LIN {X 0,Y 229.59,Z 265.503,A -85,B 0,C 180,E1 -20151.196,E2 -20151.196} C_VEL
LIN {X 0,Y 229.22,Z 263.63,A -85,B 0,C 180,E1 -20152.955,E2 -20152.955} C_VEL
LIN {X 0,Y 228.29,Z 260.05,A -85,B 0,C 180,E1 -20156.691,E2 -20156.691} C_VEL
LIN {X 0,Y 228.555,Z 260.016,A -85,B 0,C 180,E1 -20158.238,E2 -20158.238} C_VEL
LIN {X 0,Y 228.555,Z 260.014,A -85,B 0,C 180,E1 -20161.762,E2 -20161.762} C_VEL
LIN {X 0,Y 228.313,Z 260.047,A -85,B 0,C 180,E1 -20167.073,E2 -20167.073} C_VEL
LIN {X 0,Y 228.147,Z 260.063,A -85,B 0,C 180,E1 -20170.651,E2 -20170.651} C_VEL
LIN {X 0,Y 228.066,Z 260.074,A -85,B 0,C 180,E1 -20174.272,E2 -20174.272} C_VEL
LIN {X 0,Y 228.004,Z 260.082,A -85,B 0,C 180,E1 -20177.953,E2 -20177.953} C_VEL
LIN {X 0,Y 227.918,Z 260.094,A -85,B 0,C 180,E1 -20182.321,E2 -20182.321} C_VEL
LIN {X 0,Y 227.944,Z 260.087,A -85,B 0,C 180,E1 -20186.603,E2 -20186.603} C_VEL
LIN {X 0,Y 227.91,Z 260.093,A -85,B 0,C 180,E1 -20190.296,E2 -20190.296} C_VEL
LIN {X 0,Y 227.889,Z 260.097,A -85,B 0,C 180,E1 -20193.718,E2 -20193.718} C_VEL
LIN {X 0,Y 227.86,Z 260.1,A -85,B 0,C 180,E1 -20198.088,E2 -20198.088} C_VEL
LIN {X 0,Y 227.945,Z 260.09,A -85,B 0,C 180,E1 -20202.711,E2 -20202.711} C_VEL
LIN {X 0,Y 228.096,Z 260.26,A -85,B 0,C 180,E1 -20204.606,E2 -20204.606} C_VEL
LIN {X 0,Y 228.501,Z 262.622,A -85,B 0,C 180,E1 -20206.87,E2 -20206.87} C_VEL
LIN {X 0,Y 230.282,Z 270.126,A -85,B 0,C 180,E1 -20211.134,E2 -20211.134} C_VEL
LIN {X 0,Y 230.396,Z 272.05,A -85,B 0,C 180,E1 -20211.985,E2 -20211.985} C_VEL
LIN {X 0,Y 229.973,Z 274.309,A -85,B 0,C 180,E1 -20212.782,E2 -20212.782} C_VEL
LIN {X 0,Y 228.181,Z 279.291,A -85,B 0,C 180,E1 -20214.258,E2 -20214.258} C_VEL
LIN {X 0,Y 225.385,Z 287.27,A -85,B 0,C 180,E1 -20216.474,E2 -20216.474} C_VEL
LIN {X 0,Y 225.099,Z 289.77,A -85,B 0,C 180,E1 -20217.278,E2 -20217.278} C_VEL
LIN {X 0,Y 225.285,Z 297.17,A -85,B 0,C 180,E1 -20219.681,E2 -20219.681} C_VEL
LIN {X 0,Y 228.899,Z 309.726,A -85,B 0,C 180,E1 -20221.127,E2 -20221.127} C_VEL
LIN {X 0,Y 230.455,Z 318.269,A -85,B 0,C 180,E1 -20222.176,E2 -20222.176} C_VEL
LIN {X 0,Y 230.206,Z 328.596,A -85,B 0,C 180,E1 -20223.391,E2 -20223.391} C_VEL
LIN {X 0,Y 229.898,Z 337.162,A -85,B 0,C 180,E1 -20224.661,E2 -20224.661} C_VEL
LIN {X 0,Y 229.393,Z 343.849,A -85,B 0,C 180,E1 -20225.809,E2 -20225.809} C_VEL
LIN {X 0,Y 227.633,Z 351.72,A -85,B 0,C 180,E1 -20227.299,E2 -20227.299} C_VEL
LIN {X 0,Y 225.585,Z 359.464,A -85,B 0,C 180,E1 -20229.101,E2 -20229.101} C_VEL
LIN {X 0,Y 224.128,Z 365.266,A -85,B 0,C 180,E1 -20230.777,E2 -20230.777} C_VEL
LIN {X 0,Y 222.433,Z 371.587,A -85,B 0,C 180,E1 -20233.007,E2 -20233.007} C_VEL
LIN {X 0,Y 220.953,Z 376.675,A -85,B 0,C 180,E1 -20235.259,E2 -20235.259} C_VEL
LIN {X 0,Y 219.787,Z 381.363,A -85,B 0,C 180,E1 -20238.004,E2 -20238.004} C_VEL
LIN {X 0,Y 219.081,Z 384.647,A -85,B 0,C 180,E1 -20240.77,E2 -20240.77} C_VEL
LIN {X 0,Y 218.848,Z 386.24,A -85,B 0,C 180,E1 -20242.62,E2 -20242.62} C_VEL
LIN {X 0,Y 218.718,Z 387.462,A -85,B 0,C 180,E1 -20244.946,E2 -20244.946} C_VEL
LIN {X 0,Y 218.899,Z 387.78,A -85,B 0,C 180,E1 -20248.16,E2 -20248.16} C_VEL
LIN {X 0,Y 219.007,Z 387.299,A -85,B 0,C 180,E1 -20250,E2 -20250} C_VEL
LIN {X 0,Y 219.025,Z 386.314,A -85,B 0,C 180,E1 -20251.839,E2 -20251.839} C_VEL
LIN {X 0,Y 218.977,Z 384.863,A -85,B 0,C 180,E1 -20253.681,E2 -20253.681} C_VEL
LIN {X 0,Y 218.888,Z 386.594,A -85,B 0,C 180,E1 -20257.379,E2 -20257.379} C_VEL
LIN {X 0,Y 219.575,Z 386.929,A -85,B 0,C 180,E1 -20261.072,E2 -20261.072} C_VEL
LIN {X 0,Y 221.154,Z 385.921,A -85,B 0,C 180,E1 -20264.728,E2 -20264.728} C_VEL
LIN {X 0,Y 224.036,Z 383.598,A -85,B 0,C 180,E1 -20268.283,E2 -20268.283} C_VEL
LIN {X 0,Y 227.711,Z 379.914,A -85,B 0,C 180,E1 -20271.738,E2 -20271.738} C_VEL
LIN {X 0,Y 232.452,Z 374.872,A -85,B 0,C 180,E1 -20275.042,E2 -20275.042} C_VEL
LIN {X 0,Y 238.466,Z 368.336,A -85,B 0,C 180,E1 -20278.135,E2 -20278.135} C_VEL
LIN {X 0,Y 245.331,Z 360.115,A -85,B 0,C 180,E1 -20281.041,E2 -20281.041} C_VEL
LIN {X 0,Y 247.83,Z 356.7,A -85,B 0,C 180,E1 -20282.122,E2 -20282.122} C_VEL
LIN {X 0,Y 250.643,Z 351.199,A -85,B 0,C 180,E1 -20284.112,E2 -20284.112} C_VEL
LIN {X 0,Y 253.194,Z 344.707,A -85,B 0,C 180,E1 -20286.639,E2 -20286.639} C_VEL
LIN {X 0,Y 255.221,Z 338.662,A -85,B 0,C 180,E1 -20289.298,E2 -20289.298} C_VEL
LIN {X 0,Y 256.199,Z 335.187,A -85,B 0,C 180,E1 -20291.176,E2 -20291.176} C_VEL
LIN {X 0,Y 256.438,Z 333.729,A -85,B 0,C 180,E1 -20292.271,E2 -20292.271} C_VEL
LIN {X 0,Y 256.512,Z 331.788,A -85,B 0,C 180,E1 -20294.573,E2 -20294.573} C_VEL
LIN {X 0,Y 256.711,Z 330.528,A -85,B 0,C 180,E1 -20297.663,E2 -20297.663} C_VEL
LIN {X 0,Y 257.03,Z 330.502,A -85,B 0,C 180,E1 -20299.962,E2 -20299.962} C_VEL
LIN {X 0,Y 257.237,Z 331.647,A -85,B 0,C 180,E1 -20302.403,E2 -20302.403} C_VEL
LIN {X 0,Y 257.278,Z 333.985,A -85,B 0,C 180,E1 -20305.036,E2 -20305.036} C_VEL
LIN {X 0,Y 256.953,Z 336.363,A -85,B 0,C 180,E1 -20306.837,E2 -20306.837} C_VEL
LIN {X 0,Y 256.352,Z 339.157,A -85,B 0,C 180,E1 -20308.608,E2 -20308.608} C_VEL
LIN {X 0,Y 255.812,Z 340.134,A -85,B 0,C 180,E1 -20309.005,E2 -20309.005} C_VEL
LIN {X 0,Y 249.23,Z 347.794,A -85,B 0,C 180,E1 -20311.355,E2 -20311.355} C_VEL
LIN {X 0,Y 244.122,Z 353.199,A -85,B 0,C 180,E1 -20313.498,E2 -20313.498} C_VEL
LIN {X 0,Y 237.984,Z 358.947,A -85,B 0,C 180,E1 -20316.505,E2 -20316.505} C_VEL
LIN {X 0,Y 233.908,Z 362.242,A -85,B 0,C 180,E1 -20318.866,E2 -20318.866} C_VEL
LIN {X 0,Y 229.169,Z 365.414,A -85,B 0,C 180,E1 -20322.141,E2 -20322.141} C_VEL
LIN {X 0,Y 225.4,Z 367.13,A -85,B 0,C 180,E1 -20325.556,E2 -20325.556} C_VEL
LIN {X 0,Y 223.711,Z 367.493,A -85,B 0,C 180,E1 -20327.296,E2 -20327.296} C_VEL
LIN {X 0,Y 221.617,Z 367.146,A -85,B 0,C 180,E1 -20330.877,E2 -20330.877} C_VEL
LIN {X 0,Y 220.129,Z 365.421,A -85,B 0,C 180,E1 -20334.504,E2 -20334.504} C_VEL
LIN {X 0,Y 219.102,Z 362.21,A -85,B 0,C 180,E1 -20338.162,E2 -20338.162} C_VEL
LIN {X 0,Y 218.911,Z 357.473,A -85,B 0,C 180,E1 -20341.84,E2 -20341.84} C_VEL
LIN {X 0,Y 218.884,Z 352.437,A -85,B 0,C 180,E1 -20344.746,E2 -20344.746} C_VEL
LIN {X 0,Y 219.258,Z 345.516,A -85,B 0,C 180,E1 -20347.903,E2 -20347.903} C_VEL
LIN {X 0,Y 219.791,Z 338.239,A -85,B 0,C 180,E1 -20350.595,E2 -20350.595} C_VEL
LIN {X 0,Y 220.562,Z 329.134,A -85,B 0,C 180,E1 -20353.357,E2 -20353.357} C_VEL
LIN {X 0,Y 221.665,Z 318.962,A -85,B 0,C 180,E1 -20355.871,E2 -20355.871} C_VEL
LIN {X 0,Y 222.811,Z 307.745,A -85,B 0,C 180,E1 -20358.149,E2 -20358.149} C_VEL
LIN {X 0,Y 224.156,Z 295.298,A -85,B 0,C 180,E1 -20360.175,E2 -20360.175} C_VEL
LIN {X 0,Y 224.4,Z 292.082,A -85,B 0,C 180,E1 -20360.631,E2 -20360.631} C_VEL
LIN {X 0,Y 222.196,Z 278.963,A -85,B 0,C 180,E1 -20362.307,E2 -20362.307} C_VEL
LIN {X 0,Y 219.935,Z 265.484,A -85,B 0,C 180,E1 -20363.663,E2 -20363.663} C_VEL
LIN {X 0,Y 219.354,Z 261.163,A -85,B 0,C 180,E1 -20364.07,E2 -20364.07} C_VEL
LIN {X 0,Y 219.832,Z 261.101,A -85,B 0,C 180,E1 -20368.656,E2 -20368.656} C_VEL
LIN {X 0,Y 220.291,Z 261.043,A -85,B 0,C 180,E1 -20372.845,E2 -20372.845} C_VEL
LIN {X 0,Y 220.71,Z 260.994,A -85,B 0,C 180,E1 -20377.243,E2 -20377.243} C_VEL
LIN {X 0,Y 220.775,Z 260.981,A -85,B 0,C 180,E1 -20380.181,E2 -20380.181} C_VEL
LIN {X 0,Y 220.769,Z 260.985,A -85,B 0,C 180,E1 -20384.456,E2 -20384.456} C_VEL
LIN {X 0,Y 220.761,Z 260.983,A -85,B 0,C 180,E1 -20388.045,E2 -20388.045} C_VEL
LIN {X 0,Y 220.827,Z 260.978,A -85,B 0,C 180,E1 -20392.793,E2 -20392.793} C_VEL
LIN {X 0,Y 220.815,Z 260.978,A -85,B 0,C 180,E1 -20397.243,E2 -20397.243} C_VEL
LIN {X 0,Y 220.809,Z 260.979,A -85,B 0,C 180,E1 -20401.482,E2 -20401.482} C_VEL
LIN {X 0,Y 220.854,Z 260.973,A -85,B 0,C 180,E1 -20405.563,E2 -20405.563} C_VEL
LIN {X 0,Y 220.891,Z 260.969,A -85,B 0,C 180,E1 -20409.513,E2 -20409.513} C_VEL
LIN {X 0,Y 221.02,Z 260.948,A -85,B 0,C 180,E1 -20413.37,E2 -20413.37} C_VEL
LIN {X 0,Y 221.085,Z 260.946,A -85,B 0,C 180,E1 -20419.004,E2 -20419.004} C_VEL
LIN {X 0,Y 221.245,Z 260.927,A -85,B 0,C 180,E1 -20422.7,E2 -20422.7} C_VEL
LIN {X 0,Y 221.488,Z 260.898,A -85,B 0,C 180,E1 -20429.091,E2 -20429.091} C_VEL
LIN {X 0,Y 221.548,Z 261.06,A -85,B 0,C 180,E1 -20430,E2 -20430} C_VEL
LIN {X 0,Y 221.881,Z 264.958,A -85,B 0,C 180,E1 -20432.723,E2 -20432.723} C_VEL
LIN {X 0,Y 221.791,Z 268.968,A -85,B 0,C 180,E1 -20435.455,E2 -20435.455} C_VEL
LIN {X 0,Y 221.3,Z 275.909,A -85,B 0,C 180,E1 -20440.102,E2 -20440.102} C_VEL
LIN {X 0,Y 220.873,Z 282.219,A -85,B 0,C 180,E1 -20444.276,E2 -20444.276} C_VEL
LIN {X 0,Y 222.943,Z 293.041,A -85,B 0,C 180,E1 -20445.191,E2 -20445.191} C_VEL
LIN {X 0,Y 224.555,Z 303.788,A -85,B 0,C 180,E1 -20446.36,E2 -20446.36} C_VEL
LIN {X 0,Y 225.741,Z 313.184,A -85,B 0,C 180,E1 -20447.671,E2 -20447.671} C_VEL
LIN {X 0,Y 224.619,Z 322.5,A -85,B 0,C 180,E1 -20449.179,E2 -20449.179} C_VEL
LIN {X 0,Y 223.529,Z 330.156,A -85,B 0,C 180,E1 -20450.714,E2 -20450.714} C_VEL
LIN {X 0,Y 222.436,Z 337.562,A -85,B 0,C 180,E1 -20452.537,E2 -20452.537} C_VEL
LIN {X 0,Y 221.49,Z 343.632,A -85,B 0,C 180,E1 -20454.362,E2 -20454.362} C_VEL
LIN {X 0,Y 220.462,Z 350.189,A -85,B 0,C 180,E1 -20456.797,E2 -20456.797} C_VEL
LIN {X 0,Y 219.652,Z 355.46,A -85,B 0,C 180,E1 -20459.4,E2 -20459.4} C_VEL
LIN {X 0,Y 219.037,Z 359.351,A -85,B 0,C 180,E1 -20461.966,E2 -20461.966} C_VEL
LIN {X 0,Y 218.799,Z 361.066,A -85,B 0,C 180,E1 -20463.369,E2 -20463.369} C_VEL
LIN {X 0,Y 218.61,Z 362.855,A -85,B 0,C 180,E1 -20465.357,E2 -20465.357} C_VEL
LIN {X 0,Y 218.638,Z 364.15,A -85,B 0,C 180,E1 -20467.643,E2 -20467.643} C_VEL
LIN {X 0,Y 218.886,Z 364.671,A -85,B 0,C 180,E1 -20469.953,E2 -20469.953} C_VEL
LIN {X 0,Y 219.44,Z 364.308,A -85,B 0,C 180,E1 -20472.555,E2 -20472.555} C_VEL
LIN {X 0,Y 220.372,Z 362.667,A -85,B 0,C 180,E1 -20475.443,E2 -20475.443} C_VEL
LIN {X 0,Y 221.05,Z 361.34,A -85,B 0,C 180,E1 -20476.992,E2 -20476.992} C_VEL
LIN {X 0,Y 222.318,Z 358.407,A -85,B 0,C 180,E1 -20479.349,E2 -20479.349} C_VEL
LIN {X 0,Y 223.916,Z 354.408,A -85,B 0,C 180,E1 -20481.69,E2 -20481.69} C_VEL
LIN {X 0,Y 225.719,Z 349.165,A -85,B 0,C 180,E1 -20484.051,E2 -20484.051} C_VEL
LIN {X 0,Y 227.969,Z 342.698,A -85,B 0,C 180,E1 -20486.295,E2 -20486.295} C_VEL
LIN {X 0,Y 230.573,Z 334.068,A -85,B 0,C 180,E1 -20488.59,E2 -20488.59} C_VEL
LIN {X 0,Y 232.363,Z 327.05,A -85,B 0,C 180,E1 -20490.063,E2 -20490.063} C_VEL
LIN {X 0,Y 233.04,Z 323.859,A -85,B 0,C 180,E1 -20490.656,E2 -20490.656} C_VEL
LIN {X 0,Y 232.499,Z 314.637,A -85,B 0,C 180,E1 -20492.501,E2 -20492.501} C_VEL
LIN {X 0,Y 230.769,Z 304.608,A -85,B 0,C 180,E1 -20494.279,E2 -20494.279} C_VEL
LIN {X 0,Y 228.071,Z 294.64,A -85,B 0,C 180,E1 -20495.917,E2 -20495.917} C_VEL
LIN {X 0,Y 224.258,Z 284.286,A -85,B 0,C 180,E1 -20497.546,E2 -20497.546} C_VEL
LIN {X 0,Y 224.75,Z 279.926,A -85,B 0,C 180,E1 -20500.832,E2 -20500.832} C_VEL
LIN {X 0,Y 224.337,Z 275.444,A -85,B 0,C 180,E1 -20504.556,E2 -20504.556} C_VEL
LIN {X 0,Y 223.778,Z 272.373,A -85,B 0,C 180,E1 -20507.3,E2 -20507.3} C_VEL
LIN {X 0,Y 223.061,Z 268.507,A -85,B 0,C 180,E1 -20510.936,E2 -20510.936} C_VEL
LIN {X 0,Y 222.706,Z 266.592,A -85,B 0,C 180,E1 -20512.748,E2 -20512.748} C_VEL
LIN {X 0,Y 221.517,Z 260.891,A -85,B 0,C 180,E1 -20519.091,E2 -20519.091} C_VEL
LIN {X 0,Y 221.512,Z 260.891,A -85,B 0,C 180,E1 -20521.818,E2 -20521.818} C_VEL
LIN {X 0,Y 221.249,Z 260.927,A -85,B 0,C 180,E1 -20527.3,E2 -20527.3} C_VEL
LIN {X 0,Y 221.069,Z 260.944,A -85,B 0,C 180,E1 -20530.996,E2 -20530.996} C_VEL
LIN {X 0,Y 220.998,Z 260.958,A -85,B 0,C 180,E1 -20534.738,E2 -20534.738} C_VEL
LIN {X 0,Y 220.922,Z 260.962,A -85,B 0,C 180,E1 -20538.549,E2 -20538.549} C_VEL
LIN {X 0,Y 220.886,Z 260.972,A -85,B 0,C 180,E1 -20542.676,E2 -20542.676} C_VEL
LIN {X 0,Y 220.887,Z 260.966,A -85,B 0,C 180,E1 -20547.016,E2 -20547.016} C_VEL
LIN {X 0,Y 220.864,Z 260.974,A -85,B 0,C 180,E1 -20550.778,E2 -20550.778} C_VEL
LIN {X 0,Y 220.815,Z 260.974,A -85,B 0,C 180,E1 -20554.952,E2 -20554.952} C_VEL
LIN {X 0,Y 220.839,Z 260.971,A -85,B 0,C 180,E1 -20557.288,E2 -20557.288} C_VEL
LIN {X 0,Y 220.891,Z 260.976,A -85,B 0,C 180,E1 -20562.482,E2 -20562.482} C_VEL
LIN {X 0,Y 222.255,Z 265.363,A -85,B 0,C 180,E1 -20565.92,E2 -20565.92} C_VEL
LIN {X 0,Y 224.08,Z 273.009,A -85,B 0,C 180,E1 -20570.459,E2 -20570.459} C_VEL
LIN {X 0,Y 224.711,Z 276.447,A -85,B 0,C 180,E1 -20572.177,E2 -20572.177} C_VEL
LIN {X 0,Y 225.03,Z 279.753,A -85,B 0,C 180,E1 -20573.602,E2 -20573.602} C_VEL
LIN {X 0,Y 225.099,Z 289.77,A -85,B 0,C 180,E1 -20577.278,E2 -20577.278} C_VEL
LIN {X 0,Y 224.986,Z 292.435,A -85,B 0,C 180,E1 -20578.005,E2 -20578.005} C_VEL
LIN {X 0,Y 224.544,Z 297.298,A -85,B 0,C 180,E1 -20578.85,E2 -20578.85} C_VEL
LIN {X 0,Y 224.008,Z 302.701,A -85,B 0,C 180,E1 -20579.48,E2 -20579.48} C_VEL
LIN {X 0,Y 223.742,Z 314.157,A -85,B 0,C 180,E1 -20580.57,E2 -20580.57} C_VEL
LIN {X 0,Y 224.211,Z 317.803,A -85,B 0,C 180,E1 -20581.01,E2 -20581.01} C_VEL
LIN {X 0,Y 224.372,Z 322.343,A -85,B 0,C 180,E1 -20581.586,E2 -20581.586} C_VEL
LIN {X 0,Y 223.972,Z 331.653,A -85,B 0,C 180,E1 -20582.819,E2 -20582.819} C_VEL
LIN {X 0,Y 223.313,Z 342.331,A -85,B 0,C 180,E1 -20584.609,E2 -20584.609} C_VEL
LIN {X 0,Y 221.709,Z 350.352,A -85,B 0,C 180,E1 -20586.161,E2 -20586.161} C_VEL
LIN {X 0,Y 219.54,Z 358.084,A -85,B 0,C 180,E1 -20587.955,E2 -20587.955} C_VEL
LIN {X 0,Y 217.789,Z 364.251,A -85,B 0,C 180,E1 -20589.725,E2 -20589.725} C_VEL
LIN {X 0,Y 216.004,Z 370.605,A -85,B 0,C 180,E1 -20591.995,E2 -20591.995} C_VEL
LIN {X 0,Y 214.731,Z 374.817,A -85,B 0,C 180,E1 -20593.847,E2 -20593.847} C_VEL
LIN {X 0,Y 213.584,Z 378.333,A -85,B 0,C 180,E1 -20595.713,E2 -20595.713} C_VEL
LIN {X 0,Y 212.494,Z 382.423,A -85,B 0,C 180,E1 -20598.554,E2 -20598.554} C_VEL
LIN {X 0,Y 212.05,Z 384.441,A -85,B 0,C 180,E1 -20600.461,E2 -20600.461} C_VEL
LIN {X 0,Y 211.765,Z 385.958,A -85,B 0,C 180,E1 -20602.372,E2 -20602.372} C_VEL
LIN {X 0,Y 211.626,Z 387.17,A -85,B 0,C 180,E1 -20605.062,E2 -20605.062} C_VEL
LIN {X 0,Y 211.823,Z 387.355,A -85,B 0,C 180,E1 -20608.099,E2 -20608.099} C_VEL
LIN {X 0,Y 211.93,Z 386.805,A -85,B 0,C 180,E1 -20610,E2 -20610} C_VEL
LIN {X 0,Y 211.952,Z 385.75,A -85,B 0,C 180,E1 -20611.901,E2 -20611.901} C_VEL
LIN {X 0,Y 211.936,Z 383.916,A -85,B 0,C 180,E1 -20614.032,E2 -20614.032} C_VEL
LIN {X 0,Y 211.863,Z 385.771,A -85,B 0,C 180,E1 -20617.625,E2 -20617.625} C_VEL
LIN {X 0,Y 212.602,Z 386.405,A -85,B 0,C 180,E1 -20621.44,E2 -20621.44} C_VEL
LIN {X 0,Y 214.284,Z 385.676,A -85,B 0,C 180,E1 -20625.212,E2 -20625.212} C_VEL
LIN {X 0,Y 217.288,Z 383.657,A -85,B 0,C 180,E1 -20628.872,E2 -20628.872} C_VEL
LIN {X 0,Y 221.159,Z 380.358,A -85,B 0,C 180,E1 -20632.417,E2 -20632.417} C_VEL
LIN {X 0,Y 226.105,Z 375.753,A -85,B 0,C 180,E1 -20635.796,E2 -20635.796} C_VEL
LIN {X 0,Y 232.331,Z 369.655,A -85,B 0,C 180,E1 -20638.947,E2 -20638.947} C_VEL
LIN {X 0,Y 239.46,Z 362.026,A -85,B 0,C 180,E1 -20641.89,E2 -20641.89} C_VEL
LIN {X 0,Y 242.128,Z 358.813,A -85,B 0,C 180,E1 -20642.973,E2 -20642.973} C_VEL
LIN {X 0,Y 245.144,Z 353.691,A -85,B 0,C 180,E1 -20644.987,E2 -20644.987} C_VEL
LIN {X 0,Y 247.873,Z 347.886,A -85,B 0,C 180,E1 -20647.449,E2 -20647.449} C_VEL
LIN {X 0,Y 249.775,Z 343.412,A -85,B 0,C 180,E1 -20649.546,E2 -20649.546} C_VEL
LIN {X 0,Y 250.885,Z 340.5,A -85,B 0,C 180,E1 -20651.17,E2 -20651.17} C_VEL
LIN {X 0,Y 251.289,Z 339.097,A -85,B 0,C 180,E1 -20652.163,E2 -20652.163} C_VEL
LIN {X 0,Y 251.525,Z 337.796,A -85,B 0,C 180,E1 -20653.408,E2 -20653.408} C_VEL
LIN {X 0,Y 251.718,Z 335.986,A -85,B 0,C 180,E1 -20656.546,E2 -20656.546} C_VEL
LIN {X 0,Y 251.971,Z 335.535,A -85,B 0,C 180,E1 -20658.859,E2 -20658.859} C_VEL
LIN {X 0,Y 252.16,Z 336.071,A -85,B 0,C 180,E1 -20661.297,E2 -20661.297} C_VEL
LIN {X 0,Y 252.015,Z 337.874,A -85,B 0,C 180,E1 -20663.973,E2 -20663.973} C_VEL
LIN {X 0,Y 251.962,Z 338.788,A -85,B 0,C 180,E1 -20664.96,E2 -20664.96} C_VEL
LIN {X 0,Y 250.897,Z 342.541,A -85,B 0,C 180,E1 -20667.845,E2 -20667.845} C_VEL
LIN {X 0,Y 250.156,Z 343.516,A -85,B 0,C 180,E1 -20668.223,E2 -20668.223} C_VEL
LIN {X 0,Y 243.383,Z 350.626,A -85,B 0,C 180,E1 -20670.601,E2 -20670.601} C_VEL
LIN {X 0,Y 236.426,Z 357.041,A -85,B 0,C 180,E1 -20673.52,E2 -20673.52} C_VEL
LIN {X 0,Y 230.233,Z 361.954,A -85,B 0,C 180,E1 -20676.62,E2 -20676.62} C_VEL
LIN {X 0,Y 224.893,Z 365.367,A -85,B 0,C 180,E1 -20679.894,E2 -20679.894} C_VEL
LIN {X 0,Y 220.464,Z 367.42,A -85,B 0,C 180,E1 -20683.327,E2 -20683.327} C_VEL
LIN {X 0,Y 216.847,Z 368.148,A -85,B 0,C 180,E1 -20686.887,E2 -20686.887} C_VEL
LIN {X 0,Y 214.638,Z 367.439,A -85,B 0,C 180,E1 -20690.577,E2 -20690.577} C_VEL
LIN {X 0,Y 213.083,Z 365.383,A -85,B 0,C 180,E1 -20694.322,E2 -20694.322} C_VEL
LIN {X 0,Y 212.033,Z 361.897,A -85,B 0,C 180,E1 -20698.101,E2 -20698.101} C_VEL
LIN {X 0,Y 211.846,Z 356.788,A -85,B 0,C 180,E1 -20701.901,E2 -20701.901} C_VEL
LIN {X 0,Y 211.86,Z 350.903,A -85,B 0,C 180,E1 -20705.206,E2 -20705.206} C_VEL
LIN {X 0,Y 212.318,Z 343.249,A -85,B 0,C 180,E1 -20708.567,E2 -20708.567} C_VEL
LIN {X 0,Y 212.903,Z 335.182,A -85,B 0,C 180,E1 -20711.424,E2 -20711.424} C_VEL
LIN {X 0,Y 213.879,Z 325.357,A -85,B 0,C 180,E1 -20714.268,E2 -20714.268} C_VEL
LIN {X 0,Y 215.059,Z 314.339,A -85,B 0,C 180,E1 -20716.86,E2 -20716.86} C_VEL
LIN {X 0,Y 216.162,Z 303.326,A -85,B 0,C 180,E1 -20718.974,E2 -20718.974} C_VEL
LIN {X 0,Y 217.29,Z 292.635,A -85,B 0,C 180,E1 -20720.656,E2 -20720.656} C_VEL
LIN {X 0,Y 215.009,Z 278.935,A -85,B 0,C 180,E1 -20722.46,E2 -20722.46} C_VEL
LIN {X 0,Y 212.768,Z 265.232,A -85,B 0,C 180,E1 -20723.869,E2 -20723.869} C_VEL
LIN {X 0,Y 212.309,Z 262.041,A -85,B 0,C 180,E1 -20724.183,E2 -20724.183} C_VEL
LIN {X 0,Y 212.637,Z 261.997,A -85,B 0,C 180,E1 -20727.563,E2 -20727.563} C_VEL
LIN {X 0,Y 213.107,Z 261.939,A -85,B 0,C 180,E1 -20731.848,E2 -20731.848} C_VEL
LIN {X 0,Y 213.415,Z 261.896,A -85,B 0,C 180,E1 -20734.585,E2 -20734.585} C_VEL
LIN {X 0,Y 213.667,Z 261.87,A -85,B 0,C 180,E1 -20738.679,E2 -20738.679} C_VEL
LIN {X 0,Y 213.706,Z 261.863,A -85,B 0,C 180,E1 -20741.127,E2 -20741.127} C_VEL
LIN {X 0,Y 213.706,Z 261.865,A -85,B 0,C 180,E1 -20743.679,E2 -20743.679} C_VEL
LIN {X 0,Y 213.705,Z 261.864,A -85,B 0,C 180,E1 -20746.345,E2 -20746.345} C_VEL
LIN {X 0,Y 213.71,Z 261.867,A -85,B 0,C 180,E1 -20749.146,E2 -20749.146} C_VEL
LIN {X 0,Y 213.744,Z 261.858,A -85,B 0,C 180,E1 -20753.711,E2 -20753.711} C_VEL
LIN {X 0,Y 213.761,Z 261.858,A -85,B 0,C 180,E1 -20758.261,E2 -20758.261} C_VEL
LIN {X 0,Y 213.793,Z 261.856,A -85,B 0,C 180,E1 -20762.598,E2 -20762.598} C_VEL
LIN {X 0,Y 213.815,Z 261.848,A -85,B 0,C 180,E1 -20766.978,E2 -20766.978} C_VEL
LIN {X 0,Y 213.947,Z 261.829,A -85,B 0,C 180,E1 -20772.803,E2 -20772.803} C_VEL
LIN {X 0,Y 213.956,Z 261.831,A -85,B 0,C 180,E1 -20776.706,E2 -20776.706} C_VEL
LIN {X 0,Y 214.139,Z 261.813,A -85,B 0,C 180,E1 -20780.555,E2 -20780.555} C_VEL
LIN {X 0,Y 214.074,Z 261.82,A -85,B 0,C 180,E1 -20784.347,E2 -20784.347} C_VEL
LIN {X 0,Y 214.459,Z 261.774,A -85,B 0,C 180,E1 -20789.354,E2 -20789.354} C_VEL
LIN {X 0,Y 214.916,Z 265.147,A -85,B 0,C 180,E1 -20791.874,E2 -20791.874} C_VEL
LIN {X 0,Y 214.874,Z 269.221,A -85,B 0,C 180,E1 -20794.69,E2 -20794.69} C_VEL
LIN {X 0,Y 214.363,Z 276.197,A -85,B 0,C 180,E1 -20799.435,E2 -20799.435} C_VEL
LIN {X 0,Y 213.893,Z 282.522,A -85,B 0,C 180,E1 -20803.721,E2 -20803.721} C_VEL
LIN {X 0,Y 216.052,Z 293.799,A -85,B 0,C 180,E1 -20804.722,E2 -20804.722} C_VEL
LIN {X 0,Y 217.638,Z 304.443,A -85,B 0,C 180,E1 -20805.931,E2 -20805.931} C_VEL
LIN {X 0,Y 218.777,Z 313.762,A -85,B 0,C 180,E1 -20807.286,E2 -20807.286} C_VEL
LIN {X 0,Y 217.664,Z 323.001,A -85,B 0,C 180,E1 -20808.837,E2 -20808.837} C_VEL
LIN {X 0,Y 216.554,Z 330.493,A -85,B 0,C 180,E1 -20810.385,E2 -20810.385} C_VEL
LIN {X 0,Y 215.586,Z 337.011,A -85,B 0,C 180,E1 -20812.018,E2 -20812.018} C_VEL
LIN {X 0,Y 214.573,Z 343.258,A -85,B 0,C 180,E1 -20813.906,E2 -20813.906} C_VEL
LIN {X 0,Y 213.791,Z 348.256,A -85,B 0,C 180,E1 -20815.735,E2 -20815.735} C_VEL
LIN {X 0,Y 212.932,Z 353.424,A -85,B 0,C 180,E1 -20818.056,E2 -20818.056} C_VEL
LIN {X 0,Y 212.236,Z 357.805,A -85,B 0,C 180,E1 -20820.574,E2 -20820.574} C_VEL
LIN {X 0,Y 211.64,Z 361.828,A -85,B 0,C 180,E1 -20823.882,E2 -20823.882} C_VEL
LIN {X 0,Y 211.521,Z 364.147,A -85,B 0,C 180,E1 -20827.114,E2 -20827.114} C_VEL
LIN {X 0,Y 211.848,Z 365.069,A -85,B 0,C 180,E1 -20830.268,E2 -20830.268} C_VEL
LIN {X 0,Y 212.735,Z 364.267,A -85,B 0,C 180,E1 -20833.929,E2 -20833.929} C_VEL
LIN {X 0,Y 214.227,Z 361.709,A -85,B 0,C 180,E1 -20837.573,E2 -20837.573} C_VEL
LIN {X 0,Y 215.672,Z 358.585,A -85,B 0,C 180,E1 -20840.123,E2 -20840.123} C_VEL
LIN {X 0,Y 217.548,Z 354.118,A -85,B 0,C 180,E1 -20842.741,E2 -20842.741} C_VEL
LIN {X 0,Y 219.722,Z 348.384,A -85,B 0,C 180,E1 -20845.283,E2 -20845.283} C_VEL
LIN {X 0,Y 222.353,Z 340.871,A -85,B 0,C 180,E1 -20847.792,E2 -20847.792} C_VEL
LIN {X 0,Y 224.367,Z 334.409,A -85,B 0,C 180,E1 -20849.474,E2 -20849.474} C_VEL
LIN {X 0,Y 226.156,Z 327.805,A -85,B 0,C 180,E1 -20850.899,E2 -20850.899} C_VEL
LIN {X 0,Y 226.689,Z 324.769,A -85,B 0,C 180,E1 -20851.501,E2 -20851.501} C_VEL
LIN {X 0,Y 226.318,Z 316.583,A -85,B 0,C 180,E1 -20853.238,E2 -20853.238} C_VEL
LIN {X 0,Y 224.858,Z 307.031,A -85,B 0,C 180,E1 -20855.084,E2 -20855.084} C_VEL
LIN {X 0,Y 222.237,Z 297.121,A -85,B 0,C 180,E1 -20856.838,E2 -20856.838} C_VEL
LIN {X 0,Y 219.092,Z 288.234,A -85,B 0,C 180,E1 -20858.356,E2 -20858.356} C_VEL
LIN {X 0,Y 217.755,Z 284.674,A -85,B 0,C 180,E1 -20858.982,E2 -20858.982} C_VEL
LIN {X 0,Y 218.009,Z 281.857,A -85,B 0,C 180,E1 -20861.193,E2 -20861.193} C_VEL
LIN {X 0,Y 217.598,Z 277.436,A -85,B 0,C 180,E1 -20865.025,E2 -20865.025} C_VEL
LIN {X 0,Y 216.868,Z 273.444,A -85,B 0,C 180,E1 -20868.788,E2 -20868.788} C_VEL
LIN {X 0,Y 216.224,Z 269.691,A -85,B 0,C 180,E1 -20872.529,E2 -20872.529} C_VEL
LIN {X 0,Y 215.2,Z 264.692,A -85,B 0,C 180,E1 -20878.128,E2 -20878.128} C_VEL
LIN {X 0,Y 214.428,Z 261.774,A -85,B 0,C 180,E1 -20881.995,E2 -20881.995} C_VEL
LIN {X 0,Y 214.19,Z 261.805,A -85,B 0,C 180,E1 -20887.542,E2 -20887.542} C_VEL
LIN {X 0,Y 214.001,Z 261.825,A -85,B 0,C 180,E1 -20891.364,E2 -20891.364} C_VEL
LIN {X 0,Y 213.936,Z 261.835,A -85,B 0,C 180,E1 -20895.237,E2 -20895.237} C_VEL
LIN {X 0,Y 213.837,Z 261.844,A -85,B 0,C 180,E1 -20899.187,E2 -20899.187} C_VEL
LIN {X 0,Y 213.812,Z 261.851,A -85,B 0,C 180,E1 -20903.231,E2 -20903.231} C_VEL
LIN {X 0,Y 213.83,Z 261.846,A -85,B 0,C 180,E1 -20907.45,E2 -20907.45} C_VEL
LIN {X 0,Y 213.78,Z 261.851,A -85,B 0,C 180,E1 -20911.735,E2 -20911.735} C_VEL
LIN {X 0,Y 213.75,Z 261.858,A -85,B 0,C 180,E1 -20916.287,E2 -20916.287} C_VEL
LIN {X 0,Y 213.783,Z 262.061,A -85,B 0,C 180,E1 -20919.26,E2 -20919.26} C_VEL
LIN {X 0,Y 215.375,Z 266.051,A -85,B 0,C 180,E1 -20923.256,E2 -20923.256} C_VEL
LIN {X 0,Y 216.629,Z 270.078,A -85,B 0,C 180,E1 -20926.313,E2 -20926.313} C_VEL
LIN {X 0,Y 218.26,Z 277.369,A -85,B 0,C 180,E1 -20930.606,E2 -20930.606} C_VEL
LIN {X 0,Y 218.822,Z 282.217,A -85,B 0,C 180,E1 -20932.904,E2 -20932.904} C_VEL
LIN {X 0,Y 218.79,Z 292.32,A -85,B 0,C 180,E1 -20936.769,E2 -20936.769} C_VEL
LIN {X 0,Y 218.853,Z 296.993,A -85,B 0,C 180,E1 -20938.313,E2 -20938.313} C_VEL
LIN {X 0,Y 222.611,Z 309.553,A -85,B 0,C 180,E1 -20939.919,E2 -20939.919} C_VEL
LIN {X 0,Y 224.211,Z 317.803,A -85,B 0,C 180,E1 -20941.01,E2 -20941.01} C_VEL
LIN {X 0,Y 224.485,Z 321.293,A -85,B 0,C 180,E1 -20941.442,E2 -20941.442} C_VEL
LIN {X 0,Y 223.688,Z 326.674,A -85,B 0,C 180,E1 -20942.005,E2 -20942.005} C_VEL
LIN {X 0,Y 221.962,Z 331.976,A -85,B 0,C 180,E1 -20942.521,E2 -20942.521} C_VEL
LIN {X 0,Y 219.037,Z 339.007,A -85,B 0,C 180,E1 -20943.278,E2 -20943.278} C_VEL
LIN {X 0,Y 217.11,Z 344.043,A -85,B 0,C 180,E1 -20944,E2 -20944} C_VEL
LIN {X 0,Y 216.627,Z 345.613,A -85,B 0,C 180,E1 -20944.284,E2 -20944.284} C_VEL
LIN {X 0,Y 214.686,Z 353.032,A -85,B 0,C 180,E1 -20945.845,E2 -20945.845} C_VEL
LIN {X 0,Y 212.44,Z 360.409,A -85,B 0,C 180,E1 -20947.741,E2 -20947.741} C_VEL
LIN {X 0,Y 209.98,Z 368.468,A -85,B 0,C 180,E1 -20950.446,E2 -20950.446} C_VEL
LIN {X 0,Y 208.545,Z 372.986,A -85,B 0,C 180,E1 -20952.344,E2 -20952.344} C_VEL
LIN {X 0,Y 207.251,Z 376.775,A -85,B 0,C 180,E1 -20954.259,E2 -20954.259} C_VEL
LIN {X 0,Y 205.849,Z 381.133,A -85,B 0,C 180,E1 -20957.178,E2 -20957.178} C_VEL
LIN {X 0,Y 205.002,Z 384.245,A -85,B 0,C 180,E1 -20960.13,E2 -20960.13} C_VEL
LIN {X 0,Y 204.695,Z 385.68,A -85,B 0,C 180,E1 -20962.107,E2 -20962.107} C_VEL
LIN {X 0,Y 204.556,Z 386.865,A -85,B 0,C 180,E1 -20965.112,E2 -20965.112} C_VEL
LIN {X 0,Y 204.746,Z 386.93,A -85,B 0,C 180,E1 -20968.033,E2 -20968.033} C_VEL
LIN {X 0,Y 204.855,Z 386.305,A -85,B 0,C 180,E1 -20970,E2 -20970} C_VEL
LIN {X 0,Y 204.877,Z 385.174,A -85,B 0,C 180,E1 -20971.966,E2 -20971.966} C_VEL
LIN {X 0,Y 204.93,Z 383.007,A -85,B 0,C 180,E1 -20974.498,E2 -20974.498} C_VEL
LIN {X 0,Y 204.854,Z 384.862,A -85,B 0,C 180,E1 -20977.888,E2 -20977.888} C_VEL
LIN {X 0,Y 205.642,Z 385.756,A -85,B 0,C 180,E1 -20981.833,E2 -20981.833} C_VEL
LIN {X 0,Y 207.434,Z 385.354,A -85,B 0,C 180,E1 -20985.727,E2 -20985.727} C_VEL
LIN {X 0,Y 210.565,Z 383.693,A -85,B 0,C 180,E1 -20989.498,E2 -20989.498} C_VEL
LIN {X 0,Y 214.641,Z 380.76,A -85,B 0,C 180,E1 -20993.137,E2 -20993.137} C_VEL
LIN {X 0,Y 219.785,Z 376.532,A -85,B 0,C 180,E1 -20996.595,E2 -20996.595} C_VEL
LIN {X 0,Y 226.249,Z 370.922,A -85,B 0,C 180,E1 -20999.803,E2 -20999.803} C_VEL
LIN {X 0,Y 233.606,Z 363.869,A -85,B 0,C 180,E1 -21002.788,E2 -21002.788} C_VEL
LIN {X 0,Y 237.21,Z 359.866,A -85,B 0,C 180,E1 -21004.259,E2 -21004.259} C_VEL
LIN {X 0,Y 240.749,Z 354.221,A -85,B 0,C 180,E1 -21006.742,E2 -21006.742} C_VEL
LIN {X 0,Y 243.678,Z 348.784,A -85,B 0,C 180,E1 -21009.384,E2 -21009.384} C_VEL
LIN {X 0,Y 245.315,Z 345.455,A -85,B 0,C 180,E1 -21011.219,E2 -21011.219} C_VEL
LIN {X 0,Y 245.8,Z 344.352,A -85,B 0,C 180,E1 -21011.978,E2 -21011.978} C_VEL
LIN {X 0,Y 246.234,Z 342.944,A -85,B 0,C 180,E1 -21013.237,E2 -21013.237} C_VEL
LIN {X 0,Y 246.497,Z 341.409,A -85,B 0,C 180,E1 -21015.463,E2 -21015.463} C_VEL
LIN {X 0,Y 246.716,Z 340.599,A -85,B 0,C 180,E1 -21017.787,E2 -21017.787} C_VEL
LIN {X 0,Y 246.951,Z 340.566,A -85,B 0,C 180,E1 -21020.211,E2 -21020.211} C_VEL
LIN {X 0,Y 246.935,Z 340.879,A -85,B 0,C 180,E1 -21021.234,E2 -21021.234} C_VEL
LIN {X 0,Y 246.674,Z 342.049,A -85,B 0,C 180,E1 -21023.251,E2 -21023.251} C_VEL
LIN {X 0,Y 246.27,Z 343.695,A -85,B 0,C 180,E1 -21025.197,E2 -21025.197} C_VEL
LIN {X 0,Y 245.41,Z 345.871,A -85,B 0,C 180,E1 -21027.036,E2 -21027.036} C_VEL
LIN {X 0,Y 237.568,Z 353.341,A -85,B 0,C 180,E1 -21029.807,E2 -21029.807} C_VEL
LIN {X 0,Y 230.364,Z 359.236,A -85,B 0,C 180,E1 -21032.766,E2 -21032.766} C_VEL
LIN {X 0,Y 223.906,Z 363.657,A -85,B 0,C 180,E1 -21035.918,E2 -21035.918} C_VEL
LIN {X 0,Y 218.353,Z 366.69,A -85,B 0,C 180,E1 -21039.265,E2 -21039.265} C_VEL
LIN {X 0,Y 213.73,Z 368.336,A -85,B 0,C 180,E1 -21042.786,E2 -21042.786} C_VEL
LIN {X 0,Y 209.972,Z 368.675,A -85,B 0,C 180,E1 -21046.45,E2 -21046.45} C_VEL
LIN {X 0,Y 207.646,Z 367.661,A -85,B 0,C 180,E1 -21050.257,E2 -21050.257} C_VEL
LIN {X 0,Y 206.042,Z 365.283,A -85,B 0,C 180,E1 -21054.127,E2 -21054.127} C_VEL
LIN {X 0,Y 204.966,Z 361.439,A -85,B 0,C 180,E1 -21058.035,E2 -21058.035} C_VEL
LIN {X 0,Y 204.781,Z 356.04,A -85,B 0,C 180,E1 -21061.967,E2 -21061.967} C_VEL
LIN {X 0,Y 204.825,Z 349.887,A -85,B 0,C 180,E1 -21065.343,E2 -21065.343} C_VEL
LIN {X 0,Y 205.295,Z 341.827,A -85,B 0,C 180,E1 -21068.862,E2 -21068.862} C_VEL
LIN {X 0,Y 205.933,Z 333.352,A -85,B 0,C 180,E1 -21071.816,E2 -21071.816} C_VEL
LIN {X 0,Y 207.006,Z 323.097,A -85,B 0,C 180,E1 -21074.752,E2 -21074.752} C_VEL
LIN {X 0,Y 208.057,Z 312.626,A -85,B 0,C 180,E1 -21077.192,E2 -21077.192} C_VEL
LIN {X 0,Y 209.452,Z 299.869,A -85,B 0,C 180,E1 -21079.606,E2 -21079.606} C_VEL
LIN {X 0,Y 210.142,Z 292.571,A -85,B 0,C 180,E1 -21080.753,E2 -21080.753} C_VEL
LIN {X 0,Y 207.766,Z 278.61,A -85,B 0,C 180,E1 -21082.634,E2 -21082.634} C_VEL
LIN {X 0,Y 205.514,Z 264.434,A -85,B 0,C 180,E1 -21084.121,E2 -21084.121} C_VEL
LIN {X 0,Y 205.285,Z 262.916,A -85,B 0,C 180,E1 -21084.257,E2 -21084.257} C_VEL
LIN {X 0,Y 205.685,Z 262.863,A -85,B 0,C 180,E1 -21088.579,E2 -21088.579} C_VEL
LIN {X 0,Y 206.197,Z 262.8,A -85,B 0,C 180,E1 -21093.048,E2 -21093.048} C_VEL
LIN {X 0,Y 206.417,Z 262.771,A -85,B 0,C 180,E1 -21095.367,E2 -21095.367} C_VEL
LIN {X 0,Y 206.63,Z 262.746,A -85,B 0,C 180,E1 -21098.529,E2 -21098.529} C_VEL
LIN {X 0,Y 206.623,Z 262.747,A -85,B 0,C 180,E1 -21102.866,E2 -21102.866} C_VEL
LIN {X 0,Y 206.623,Z 262.746,A -85,B 0,C 180,E1 -21107.134,E2 -21107.134} C_VEL
LIN {X 0,Y 206.676,Z 262.741,A -85,B 0,C 180,E1 -21111.455,E2 -21111.455} C_VEL
LIN {X 0,Y 206.702,Z 262.738,A -85,B 0,C 180,E1 -21114.689,E2 -21114.689} C_VEL
LIN {X 0,Y 206.698,Z 262.736,A -85,B 0,C 180,E1 -21119.334,E2 -21119.334} C_VEL
LIN {X 0,Y 206.71,Z 262.735,A -85,B 0,C 180,E1 -21123.769,E2 -21123.769} C_VEL
LIN {X 0,Y 206.742,Z 262.73,A -85,B 0,C 180,E1 -21128.041,E2 -21128.041} C_VEL
LIN {X 0,Y 206.877,Z 262.709,A -85,B 0,C 180,E1 -21132.196,E2 -21132.196} C_VEL
LIN {X 0,Y 206.899,Z 262.712,A -85,B 0,C 180,E1 -21136.244,E2 -21136.244} C_VEL
LIN {X 0,Y 207.083,Z 262.692,A -85,B 0,C 180,E1 -21140.23,E2 -21140.23} C_VEL
LIN {X 0,Y 207.038,Z 262.697,A -85,B 0,C 180,E1 -21144.155,E2 -21144.155} C_VEL
LIN {X 0,Y 207.415,Z 262.689,A -85,B 0,C 180,E1 -21148.908,E2 -21148.908} C_VEL
LIN {X 0,Y 207.958,Z 266.764,A -85,B 0,C 180,E1 -21151.936,E2 -21151.936} C_VEL
LIN {X 0,Y 207.857,Z 270.841,A -85,B 0,C 180,E1 -21154.849,E2 -21154.849} C_VEL
LIN {X 0,Y 207.321,Z 277.927,A -85,B 0,C 180,E1 -21159.758,E2 -21159.758} C_VEL
LIN {X 0,Y 206.927,Z 282.81,A -85,B 0,C 180,E1 -21163.128,E2 -21163.128} C_VEL
LIN {X 0,Y 209.161,Z 294.585,A -85,B 0,C 180,E1 -21164.223,E2 -21164.223} C_VEL
LIN {X 0,Y 210.727,Z 305.103,A -85,B 0,C 180,E1 -21165.474,E2 -21165.474} C_VEL
LIN {X 0,Y 211.837,Z 314.323,A -85,B 0,C 180,E1 -21166.875,E2 -21166.875} C_VEL
LIN {X 0,Y 210.711,Z 323.508,A -85,B 0,C 180,E1 -21168.473,E2 -21168.473} C_VEL
LIN {X 0,Y 209.558,Z 331.131,A -85,B 0,C 180,E1 -21170.107,E2 -21170.107} C_VEL
LIN {X 0,Y 208.561,Z 337.489,A -85,B 0,C 180,E1 -21171.757,E2 -21171.757} C_VEL
LIN {X 0,Y 207.463,Z 344.112,A -85,B 0,C 180,E1 -21173.843,E2 -21173.843} C_VEL
LIN {X 0,Y 206.418,Z 350.328,A -85,B 0,C 180,E1 -21176.271,E2 -21176.271} C_VEL
LIN {X 0,Y 205.671,Z 355.005,A -85,B 0,C 180,E1 -21178.58,E2 -21178.58} C_VEL
LIN {X 0,Y 205.033,Z 358.872,A -85,B 0,C 180,E1 -21181.025,E2 -21181.025} C_VEL
LIN {X 0,Y 204.608,Z 361.63,A -85,B 0,C 180,E1 -21183.338,E2 -21183.338} C_VEL
LIN {X 0,Y 204.434,Z 363.69,A -85,B 0,C 180,E1 -21185.762,E2 -21185.762} C_VEL
LIN {X 0,Y 204.493,Z 364.971,A -85,B 0,C 180,E1 -21188.216,E2 -21188.216} C_VEL
LIN {X 0,Y 204.886,Z 365.465,A -85,B 0,C 180,E1 -21191.005,E2 -21191.005} C_VEL
LIN {X 0,Y 205.7,Z 364.785,A -85,B 0,C 180,E1 -21194.152,E2 -21194.152} C_VEL
LIN {X 0,Y 206.273,Z 364.075,A -85,B 0,C 180,E1 -21195.684,E2 -21195.684} C_VEL
LIN {X 0,Y 207.418,Z 362.091,A -85,B 0,C 180,E1 -21198.196,E2 -21198.196} C_VEL
LIN {X 0,Y 208.914,Z 359.153,A -85,B 0,C 180,E1 -21200.69,E2 -21200.69} C_VEL
LIN {X 0,Y 210.727,Z 355.145,A -85,B 0,C 180,E1 -21203.171,E2 -21203.171} C_VEL
LIN {X 0,Y 212.812,Z 349.899,A -85,B 0,C 180,E1 -21205.651,E2 -21205.651} C_VEL
LIN {X 0,Y 215.355,Z 343.326,A -85,B 0,C 180,E1 -21208.049,E2 -21208.049} C_VEL
LIN {X 0,Y 218.226,Z 334.832,A -85,B 0,C 180,E1 -21210.405,E2 -21210.405} C_VEL
LIN {X 0,Y 220.194,Z 327.973,A -85,B 0,C 180,E1 -21211.915,E2 -21211.915} C_VEL
LIN {X 0,Y 220.406,Z 322.217,A -85,B 0,C 180,E1 -21213.23,E2 -21213.23} C_VEL
LIN {X 0,Y 219.608,Z 313.668,A -85,B 0,C 180,E1 -21215.049,E2 -21215.049} C_VEL
LIN {X 0,Y 217.993,Z 305.16,A -85,B 0,C 180,E1 -21216.738,E2 -21216.738} C_VEL
LIN {X 0,Y 215.408,Z 295.985,A -85,B 0,C 180,E1 -21218.479,E2 -21218.479} C_VEL
LIN {X 0,Y 212.408,Z 288.214,A -85,B 0,C 180,E1 -21219.936,E2 -21219.936} C_VEL
LIN {X 0,Y 211.258,Z 285.116,A -85,B 0,C 180,E1 -21220.49,E2 -21220.49} C_VEL
LIN {X 0,Y 211.136,Z 281.596,A -85,B 0,C 180,E1 -21223.564,E2 -21223.564} C_VEL
LIN {X 0,Y 210.723,Z 278.46,A -85,B 0,C 180,E1 -21226.499,E2 -21226.499} C_VEL
LIN {X 0,Y 209.762,Z 272.794,A -85,B 0,C 180,E1 -21232.298,E2 -21232.298} C_VEL
LIN {X 0,Y 208.771,Z 267.801,A -85,B 0,C 180,E1 -21238.071,E2 -21238.071} C_VEL
LIN {X 0,Y 208.115,Z 264.99,A -85,B 0,C 180,E1 -21241.935,E2 -21241.935} C_VEL
LIN {X 0,Y 207.065,Z 262.689,A -85,B 0,C 180,E1 -21246.333,E2 -21246.333} C_VEL
LIN {X 0,Y 207.062,Z 262.691,A -85,B 0,C 180,E1 -21250.165,E2 -21250.165} C_VEL
LIN {X 0,Y 206.869,Z 262.712,A -85,B 0,C 180,E1 -21255.77,E2 -21255.77} C_VEL
LIN {X 0,Y 206.78,Z 262.727,A -85,B 0,C 180,E1 -21259.869,E2 -21259.869} C_VEL
LIN {X 0,Y 206.748,Z 262.727,A -85,B 0,C 180,E1 -21264.074,E2 -21264.074} C_VEL
LIN {X 0,Y 206.745,Z 262.731,A -85,B 0,C 180,E1 -21268.419,E2 -21268.419} C_VEL
LIN {X 0,Y 206.709,Z 262.733,A -85,B 0,C 180,E1 -21272.956,E2 -21272.956} C_VEL
LIN {X 0,Y 206.755,Z 262.875,A -85,B 0,C 180,E1 -21274.924,E2 -21274.924} C_VEL
LIN {X 0,Y 207.987,Z 266.006,A -85,B 0,C 180,E1 -21278.997,E2 -21278.997} C_VEL
LIN {X 0,Y 209.667,Z 270.391,A -85,B 0,C 180,E1 -21283.404,E2 -21283.404} C_VEL
LIN {X 0,Y 210.777,Z 274.23,A -85,B 0,C 180,E1 -21286.282,E2 -21286.282} C_VEL
LIN {X 0,Y 212.21,Z 280.879,A -85,B 0,C 180,E1 -21290.301,E2 -21290.301} C_VEL
LIN {X 0,Y 212.683,Z 285.359,A -85,B 0,C 180,E1 -21292.473,E2 -21292.473} C_VEL
LIN {X 0,Y 212.482,Z 295.275,A -85,B 0,C 180,E1 -21296.38,E2 -21296.38} C_VEL
LIN {X 0,Y 212.537,Z 296.79,A -85,B 0,C 180,E1 -21296.844,E2 -21296.844} C_VEL
LIN {X 0,Y 216.483,Z 309.673,A -85,B 0,C 180,E1 -21298.651,E2 -21298.651} C_VEL
LIN {X 0,Y 218.387,Z 320.524,A -85,B 0,C 180,E1 -21300.232,E2 -21300.232} C_VEL
LIN {X 0,Y 218.105,Z 329.082,A -85,B 0,C 180,E1 -21301.38,E2 -21301.38} C_VEL
LIN {X 0,Y 217.517,Z 337.267,A -85,B 0,C 180,E1 -21302.687,E2 -21302.687} C_VEL
LIN {X 0,Y 216.627,Z 345.613,A -85,B 0,C 180,E1 -21304.284,E2 -21304.284} C_VEL
LIN {X 0,Y 214.876,Z 349.35,A -85,B 0,C 180,E1 -21304.883,E2 -21304.883} C_VEL
LIN {X 0,Y 207.762,Z 357.899,A -85,B 0,C 180,E1 -21306.213,E2 -21306.213} C_VEL
LIN {X 0,Y 206.278,Z 360.138,A -85,B 0,C 180,E1 -21306.757,E2 -21306.757} C_VEL
LIN {X 0,Y 205.884,Z 361.004,A -85,B 0,C 180,E1 -21307.016,E2 -21307.016} C_VEL
LIN {X 0,Y 203.997,Z 366.775,A -85,B 0,C 180,E1 -21308.984,E2 -21308.984} C_VEL
LIN {X 0,Y 201.787,Z 373.105,A -85,B 0,C 180,E1 -21311.732,E2 -21311.732} C_VEL
LIN {X 0,Y 199.809,Z 378.323,A -85,B 0,C 180,E1 -21314.704,E2 -21314.704} C_VEL
LIN {X 0,Y 198.528,Z 382.221,A -85,B 0,C 180,E1 -21317.737,E2 -21317.737} C_VEL
LIN {X 0,Y 197.974,Z 384.06,A -85,B 0,C 180,E1 -21319.776,E2 -21319.776} C_VEL
LIN {X 0,Y 197.647,Z 385.41,A -85,B 0,C 180,E1 -21321.823,E2 -21321.823} C_VEL
LIN {X 0,Y 197.462,Z 386.58,A -85,B 0,C 180,E1 -21325.25,E2 -21325.25} C_VEL
LIN {X 0,Y 197.669,Z 386.502,A -85,B 0,C 180,E1 -21327.963,E2 -21327.963} C_VEL
LIN {X 0,Y 197.782,Z 385.803,A -85,B 0,C 180,E1 -21330,E2 -21330} C_VEL
LIN {X 0,Y 197.806,Z 384.597,A -85,B 0,C 180,E1 -21332.036,E2 -21332.036} C_VEL
LIN {X 0,Y 197.919,Z 381.988,A -85,B 0,C 180,E1 -21334.905,E2 -21334.905} C_VEL
LIN {X 0,Y 197.858,Z 383.872,A -85,B 0,C 180,E1 -21338.169,E2 -21338.169} C_VEL
LIN {X 0,Y 198.698,Z 385.071,A -85,B 0,C 180,E1 -21342.253,E2 -21342.253} C_VEL
LIN {X 0,Y 200.608,Z 384.978,A -85,B 0,C 180,E1 -21346.277,E2 -21346.277} C_VEL
LIN {X 0,Y 203.87,Z 383.63,A -85,B 0,C 180,E1 -21350.166,E2 -21350.166} C_VEL
LIN {X 0,Y 208.14,Z 381.054,A -85,B 0,C 180,E1 -21353.903,E2 -21353.903} C_VEL
LIN {X 0,Y 213.504,Z 377.251,A -85,B 0,C 180,E1 -21357.442,E2 -21357.442} C_VEL
LIN {X 0,Y 220.203,Z 372.134,A -85,B 0,C 180,E1 -21360.708,E2 -21360.708} C_VEL
LIN {X 0,Y 227.803,Z 365.591,A -85,B 0,C 180,E1 -21363.733,E2 -21363.733} C_VEL
LIN {X 0,Y 231.605,Z 361.869,A -85,B 0,C 180,E1 -21365.209,E2 -21365.209} C_VEL
LIN {X 0,Y 235.407,Z 356.641,A -85,B 0,C 180,E1 -21367.736,E2 -21367.736} C_VEL
LIN {X 0,Y 238.572,Z 351.673,A -85,B 0,C 180,E1 -21370.398,E2 -21370.398} C_VEL
LIN {X 0,Y 240.268,Z 348.701,A -85,B 0,C 180,E1 -21372.281,E2 -21372.281} C_VEL
LIN {X 0,Y 240.658,Z 347.807,A -85,B 0,C 180,E1 -21373.107,E2 -21373.107} C_VEL
LIN {X 0,Y 241.168,Z 346.041,A -85,B 0,C 180,E1 -21375.621,E2 -21375.621} C_VEL
LIN {X 0,Y 241.404,Z 345.267,A -85,B 0,C 180,E1 -21377.964,E2 -21377.964} C_VEL
LIN {X 0,Y 241.566,Z 345.186,A -85,B 0,C 180,E1 -21380.204,E2 -21380.204} C_VEL
LIN {X 0,Y 241.283,Z 345.982,A -85,B 0,C 180,E1 -21382.289,E2 -21382.289} C_VEL
LIN {X 0,Y 240.62,Z 347.754,A -85,B 0,C 180,E1 -21384.868,E2 -21384.868} C_VEL
LIN {X 0,Y 239.904,Z 349.129,A -85,B 0,C 180,E1 -21386.179,E2 -21386.179} C_VEL
LIN {X 0,Y 231.77,Z 355.978,A -85,B 0,C 180,E1 -21388.97,E2 -21388.97} C_VEL
LIN {X 0,Y 224.325,Z 361.362,A -85,B 0,C 180,E1 -21391.97,E2 -21391.97} C_VEL
LIN {X 0,Y 217.604,Z 365.303,A -85,B 0,C 180,E1 -21395.174,E2 -21395.174} C_VEL
LIN {X 0,Y 211.839,Z 367.886,A -85,B 0,C 180,E1 -21398.596,E2 -21398.596} C_VEL
LIN {X 0,Y 207.015,Z 369.184,A -85,B 0,C 180,E1 -21402.209,E2 -21402.209} C_VEL
LIN {X 0,Y 203.111,Z 369.152,A -85,B 0,C 180,E1 -21405.983,E2 -21405.983} C_VEL
LIN {X 0,Y 200.663,Z 367.763,A -85,B 0,C 180,E1 -21409.915,E2 -21409.915} C_VEL
LIN {X 0,Y 199.005,Z 365.059,A -85,B 0,C 180,E1 -21413.918,E2 -21413.918} C_VEL
LIN {X 0,Y 197.9,Z 360.909,A -85,B 0,C 180,E1 -21417.965,E2 -21417.965} C_VEL
LIN {X 0,Y 197.718,Z 355.135,A -85,B 0,C 180,E1 -21422.037,E2 -21422.037} C_VEL
LIN {X 0,Y 197.787,Z 348.947,A -85,B 0,C 180,E1 -21425.407,E2 -21425.407} C_VEL
LIN {X 0,Y 198.217,Z 341.514,A -85,B 0,C 180,E1 -21428.667,E2 -21428.667} C_VEL
LIN {X 0,Y 198.864,Z 332.942,A -85,B 0,C 180,E1 -21431.725,E2 -21431.725} C_VEL
LIN {X 0,Y 199.941,Z 322.568,A -85,B 0,C 180,E1 -21434.764,E2 -21434.764} C_VEL
LIN {X 0,Y 201.011,Z 311.927,A -85,B 0,C 180,E1 -21437.289,E2 -21437.289} C_VEL
LIN {X 0,Y 202.224,Z 300.416,A -85,B 0,C 180,E1 -21439.543,E2 -21439.543} C_VEL
LIN {X 0,Y 202.988,Z 292.735,A -85,B 0,C 180,E1 -21440.8,E2 -21440.8} C_VEL
LIN {X 0,Y 200.713,Z 279.484,A -85,B 0,C 180,E1 -21442.654,E2 -21442.654} C_VEL
LIN {X 0,Y 198.479,Z 265.251,A -85,B 0,C 180,E1 -21444.211,E2 -21444.211} C_VEL
LIN {X 0,Y 198.256,Z 263.791,A -85,B 0,C 180,E1 -21444.357,E2 -21444.357} C_VEL
LIN {X 0,Y 198.559,Z 263.75,A -85,B 0,C 180,E1 -21447.763,E2 -21447.763} C_VEL
LIN {X 0,Y 199.045,Z 263.69,A -85,B 0,C 180,E1 -21452.068,E2 -21452.068} C_VEL
LIN {X 0,Y 199.441,Z 263.641,A -85,B 0,C 180,E1 -21456.803,E2 -21456.803} C_VEL
LIN {X 0,Y 199.583,Z 263.624,A -85,B 0,C 180,E1 -21459.335,E2 -21459.335} C_VEL
LIN {X 0,Y 199.571,Z 263.623,A -85,B 0,C 180,E1 -21462.308,E2 -21462.308} C_VEL
LIN {X 0,Y 199.58,Z 263.626,A -85,B 0,C 180,E1 -21465.228,E2 -21465.228} C_VEL
LIN {X 0,Y 199.576,Z 263.622,A -85,B 0,C 180,E1 -21468.003,E2 -21468.003} C_VEL
LIN {X 0,Y 199.6,Z 263.625,A -85,B 0,C 180,E1 -21470.772,E2 -21470.772} C_VEL
LIN {X 0,Y 199.613,Z 263.621,A -85,B 0,C 180,E1 -21475.713,E2 -21475.713} C_VEL
LIN {X 0,Y 199.688,Z 263.61,A -85,B 0,C 180,E1 -21478.134,E2 -21478.134} C_VEL
LIN {X 0,Y 199.648,Z 263.617,A -85,B 0,C 180,E1 -21482.765,E2 -21482.765} C_VEL
LIN {X 0,Y 199.713,Z 263.604,A -85,B 0,C 180,E1 -21487.226,E2 -21487.226} C_VEL
LIN {X 0,Y 199.8,Z 263.592,A -85,B 0,C 180,E1 -21491.757,E2 -21491.757} C_VEL
LIN {X 0,Y 199.839,Z 263.593,A -85,B 0,C 180,E1 -21495.748,E2 -21495.748} C_VEL
LIN {X 0,Y 200.025,Z 263.572,A -85,B 0,C 180,E1 -21499.882,E2 -21499.882} C_VEL
LIN {X 0,Y 200.002,Z 263.574,A -85,B 0,C 180,E1 -21503.948,E2 -21503.948} C_VEL
LIN {X 0,Y 200.361,Z 263.722,A -85,B 0,C 180,E1 -21508.492,E2 -21508.492} C_VEL
LIN {X 0,Y 200.911,Z 266.998,A -85,B 0,C 180,E1 -21511.002,E2 -21511.002} C_VEL
LIN {X 0,Y 200.973,Z 271.121,A -85,B 0,C 180,E1 -21514.01,E2 -21514.01} C_VEL
LIN {X 0,Y 200.392,Z 278.235,A -85,B 0,C 180,E1 -21519.08,E2 -21519.08} C_VEL
LIN {X 0,Y 199.963,Z 283.166,A -85,B 0,C 180,E1 -21522.56,E2 -21522.56} C_VEL
LIN {X 0,Y 202.071,Z 294.058,A -85,B 0,C 180,E1 -21523.577,E2 -21523.577} C_VEL
LIN {X 0,Y 203.49,Z 303.44,A -85,B 0,C 180,E1 -21524.699,E2 -21524.699} C_VEL
LIN {X 0,Y 204.711,Z 313.484,A -85,B 0,C 180,E1 -21526.197,E2 -21526.197} C_VEL
LIN {X 0,Y 204.828,Z 316.339,A -85,B 0,C 180,E1 -21526.7,E2 -21526.7} C_VEL
LIN {X 0,Y 203.763,Z 323.977,A -85,B 0,C 180,E1 -21528.084,E2 -21528.084} C_VEL
LIN {X 0,Y 202.593,Z 331.409,A -85,B 0,C 180,E1 -21529.73,E2 -21529.73} C_VEL
LIN {X 0,Y 201.542,Z 337.923,A -85,B 0,C 180,E1 -21531.478,E2 -21531.478} C_VEL
LIN {X 0,Y 200.347,Z 344.852,A -85,B 0,C 180,E1 -21533.748,E2 -21533.748} C_VEL
LIN {X 0,Y 199.336,Z 350.74,A -85,B 0,C 180,E1 -21536.149,E2 -21536.149} C_VEL
LIN {X 0,Y 198.517,Z 355.752,A -85,B 0,C 180,E1 -21538.737,E2 -21538.737} C_VEL
LIN {X 0,Y 197.815,Z 359.78,A -85,B 0,C 180,E1 -21541.495,E2 -21541.495} C_VEL
LIN {X 0,Y 197.498,Z 362.033,A -85,B 0,C 180,E1 -21543.475,E2 -21543.475} C_VEL
LIN {X 0,Y 197.342,Z 364.757,A -85,B 0,C 180,E1 -21547.259,E2 -21547.259} C_VEL
LIN {X 0,Y 197.586,Z 365.647,A -85,B 0,C 180,E1 -21549.81,E2 -21549.81} C_VEL
LIN {X 0,Y 198.083,Z 365.755,A -85,B 0,C 180,E1 -21552.386,E2 -21552.386} C_VEL
LIN {X 0,Y 198.908,Z 365.028,A -85,B 0,C 180,E1 -21555.036,E2 -21555.036} C_VEL
LIN {X 0,Y 200.283,Z 363.05,A -85,B 0,C 180,E1 -21558.185,E2 -21558.185} C_VEL
LIN {X 0,Y 202.145,Z 359.788,A -85,B 0,C 180,E1 -21561.258,E2 -21561.258} C_VEL
LIN {X 0,Y 204.348,Z 355.118,A -85,B 0,C 180,E1 -21564.22,E2 -21564.22} C_VEL
LIN {X 0,Y 206.596,Z 350.016,A -85,B 0,C 180,E1 -21566.655,E2 -21566.655} C_VEL
LIN {X 0,Y 209.127,Z 343.783,A -85,B 0,C 180,E1 -21568.977,E2 -21568.977} C_VEL
LIN {X 0,Y 212.139,Z 335.3,A -85,B 0,C 180,E1 -21571.393,E2 -21571.393} C_VEL
LIN {X 0,Y 214.177,Z 328.014,A -85,B 0,C 180,E1 -21573.051,E2 -21573.051} C_VEL
LIN {X 0,Y 214.007,Z 319.889,A -85,B 0,C 180,E1 -21574.987,E2 -21574.987} C_VEL
LIN {X 0,Y 213.115,Z 312.237,A -85,B 0,C 180,E1 -21576.688,E2 -21576.688} C_VEL
LIN {X 0,Y 211.721,Z 305.318,A -85,B 0,C 180,E1 -21578.147,E2 -21578.147} C_VEL
LIN {X 0,Y 209.043,Z 296.269,A -85,B 0,C 180,E1 -21579.997,E2 -21579.997} C_VEL
LIN {X 0,Y 206.318,Z 289.344,A -85,B 0,C 180,E1 -21581.44,E2 -21581.44} C_VEL
LIN {X 0,Y 204.587,Z 285.512,A -85,B 0,C 180,E1 -21582.314,E2 -21582.314} C_VEL
LIN {X 0,Y 204.193,Z 281.581,A -85,B 0,C 180,E1 -21586.058,E2 -21586.058} C_VEL
LIN {X 0,Y 203.557,Z 277.749,A -85,B 0,C 180,E1 -21590.059,E2 -21590.059} C_VEL
LIN {X 0,Y 202.923,Z 274.237,A -85,B 0,C 180,E1 -21594.036,E2 -21594.036} C_VEL
LIN {X 0,Y 202.412,Z 271.03,A -85,B 0,C 180,E1 -21598.01,E2 -21598.01} C_VEL
LIN {X 0,Y 201.824,Z 268.267,A -85,B 0,C 180,E1 -21601.995,E2 -21601.995} C_VEL
LIN {X 0,Y 200.481,Z 265.213,A -85,B 0,C 180,E1 -21608.061,E2 -21608.061} C_VEL
LIN {X 0,Y 199.862,Z 263.585,A -85,B 0,C 180,E1 -21613.213,E2 -21613.213} C_VEL
LIN {X 0,Y 199.784,Z 263.594,A -85,B 0,C 180,E1 -21618.457,E2 -21618.457} C_VEL
LIN {X 0,Y 199.716,Z 263.603,A -85,B 0,C 180,E1 -21623.803,E2 -21623.803} C_VEL
LIN {X 0,Y 199.738,Z 263.782,A -85,B 0,C 180,E1 -21628.399,E2 -21628.399} C_VEL
LIN {X 0,Y 200.704,Z 266.474,A -85,B 0,C 180,E1 -21634.074,E2 -21634.074} C_VEL
LIN {X 0,Y 202.085,Z 269.934,A -85,B 0,C 180,E1 -21638.755,E2 -21638.755} C_VEL
LIN {X 0,Y 203.588,Z 273.761,A -85,B 0,C 180,E1 -21642.732,E2 -21642.732} C_VEL
LIN {X 0,Y 204.841,Z 278.082,A -85,B 0,C 180,E1 -21646.096,E2 -21646.096} C_VEL
LIN {X 0,Y 206.22,Z 284.92,A -85,B 0,C 180,E1 -21650.282,E2 -21650.282} C_VEL
LIN {X 0,Y 206.478,Z 288.905,A -85,B 0,C 180,E1 -21652.217,E2 -21652.217} C_VEL
LIN {X 0,Y 206.275,Z 296.329,A -85,B 0,C 180,E1 -21655.205,E2 -21655.205} C_VEL
LIN {X 0,Y 210.233,Z 309.208,A -85,B 0,C 180,E1 -21657.187,E2 -21657.187} C_VEL
LIN {X 0,Y 212.08,Z 318.758,A -85,B 0,C 180,E1 -21658.678,E2 -21658.678} C_VEL
LIN {X 0,Y 212.636,Z 324.313,A -85,B 0,C 180,E1 -21659.551,E2 -21659.551} C_VEL
LIN {X 0,Y 211.726,Z 334.811,A -85,B 0,C 180,E1 -21661.141,E2 -21661.141} C_VEL
LIN {X 0,Y 210.68,Z 344.23,A -85,B 0,C 180,E1 -21662.967,E2 -21662.967} C_VEL
LIN {X 0,Y 209.433,Z 349.8,A -85,B 0,C 180,E1 -21664.136,E2 -21664.136} C_VEL
LIN {X 0,Y 207.084,Z 357.293,A -85,B 0,C 180,E1 -21665.968,E2 -21665.968} C_VEL
LIN {X 0,Y 205.884,Z 361.004,A -85,B 0,C 180,E1 -21667.016,E2 -21667.016} C_VEL
LIN {X 0,Y 203.93,Z 364.82,A -85,B 0,C 180,E1 -21668.189,E2 -21668.189} C_VEL
LIN {X 0,Y 199.293,Z 370.487,A -85,B 0,C 180,E1 -21670.107,E2 -21670.107} C_VEL
LIN {X 0,Y 195.611,Z 374.378,A -85,B 0,C 180,E1 -21671.788,E2 -21671.788} C_VEL
LIN {X 0,Y 193.608,Z 376.987,A -85,B 0,C 180,E1 -21673.227,E2 -21673.227} C_VEL
LIN {X 0,Y 193.198,Z 377.751,A -85,B 0,C 180,E1 -21673.742,E2 -21673.742} C_VEL
LIN {X 0,Y 191.939,Z 380.957,A -85,B 0,C 180,E1 -21676.232,E2 -21676.232} C_VEL
LIN {X 0,Y 190.966,Z 383.882,A -85,B 0,C 180,E1 -21679.397,E2 -21679.397} C_VEL
LIN {X 0,Y 190.577,Z 385.143,A -85,B 0,C 180,E1 -21681.518,E2 -21681.518} C_VEL
LIN {X 0,Y 190.37,Z 386.277,A -85,B 0,C 180,E1 -21685.396,E2 -21685.396} C_VEL
LIN {X 0,Y 190.593,Z 386.072,A -85,B 0,C 180,E1 -21687.887,E2 -21687.887} C_VEL
LIN {X 0,Y 190.71,Z 385.292,A -85,B 0,C 180,E1 -21690,E2 -21690} C_VEL
LIN {X 0,Y 190.737,Z 384.001,A -85,B 0,C 180,E1 -21692.112,E2 -21692.112} C_VEL
LIN {X 0,Y 190.931,Z 381.007,A -85,B 0,C 180,E1 -21695.536,E2 -21695.536} C_VEL
LIN {X 0,Y 190.891,Z 382.799,A -85,B 0,C 180,E1 -21698.469,E2 -21698.469} C_VEL
LIN {X 0,Y 191.77,Z 384.256,A -85,B 0,C 180,E1 -21702.703,E2 -21702.703} C_VEL
LIN {X 0,Y 193.806,Z 384.474,A -85,B 0,C 180,E1 -21706.865,E2 -21706.865} C_VEL
LIN {X 0,Y 197.209,Z 383.486,A -85,B 0,C 180,E1 -21710.878,E2 -21710.878} C_VEL
LIN {X 0,Y 201.665,Z 381.295,A -85,B 0,C 180,E1 -21714.721,E2 -21714.721} C_VEL
LIN {X 0,Y 207.269,Z 377.913,A -85,B 0,C 180,E1 -21718.341,E2 -21718.341} C_VEL
LIN {X 0,Y 214.204,Z 373.24,A -85,B 0,C 180,E1 -21721.666,E2 -21721.666} C_VEL
LIN {X 0,Y 222.059,Z 367.223,A -85,B 0,C 180,E1 -21724.729,E2 -21724.729} C_VEL
LIN {X 0,Y 226.034,Z 363.783,A -85,B 0,C 180,E1 -21726.212,E2 -21726.212} C_VEL
LIN {X 0,Y 230.063,Z 358.994,A -85,B 0,C 180,E1 -21728.774,E2 -21728.774} C_VEL
LIN {X 0,Y 233.454,Z 354.444,A -85,B 0,C 180,E1 -21731.476,E2 -21731.476} C_VEL
LIN {X 0,Y 234.365,Z 353.089,A -85,B 0,C 180,E1 -21732.408,E2 -21732.408} C_VEL
LIN {X 0,Y 235.039,Z 351.917,A -85,B 0,C 180,E1 -21733.452,E2 -21733.452} C_VEL
LIN {X 0,Y 235.589,Z 350.431,A -85,B 0,C 180,E1 -21735.723,E2 -21735.723} C_VEL
LIN {X 0,Y 235.936,Z 349.525,A -85,B 0,C 180,E1 -21739.055,E2 -21739.055} C_VEL
LIN {X 0,Y 235.762,Z 349.869,A -85,B 0,C 180,E1 -21741.244,E2 -21741.244} C_VEL
LIN {X 0,Y 235.04,Z 351.179,A -85,B 0,C 180,E1 -21743.837,E2 -21743.837} C_VEL
LIN {X 0,Y 234.35,Z 352.304,A -85,B 0,C 180,E1 -21745.264,E2 -21745.264} C_VEL
LIN {X 0,Y 228.112,Z 357.067,A -85,B 0,C 180,E1 -21747.373,E2 -21747.373} C_VEL
LIN {X 0,Y 220.145,Z 362.307,A -85,B 0,C 180,E1 -21750.342,E2 -21750.342} C_VEL
LIN {X 0,Y 214.712,Z 365.295,A -85,B 0,C 180,E1 -21752.726,E2 -21752.726} C_VEL
LIN {X 0,Y 208.236,Z 368.115,A -85,B 0,C 180,E1 -21756.109,E2 -21756.109} C_VEL
LIN {X 0,Y 202.659,Z 369.631,A -85,B 0,C 180,E1 -21759.709,E2 -21759.709} C_VEL
LIN {X 0,Y 198.22,Z 369.865,A -85,B 0,C 180,E1 -21763.522,E2 -21763.522} C_VEL
LIN {X 0,Y 196.239,Z 369.512,A -85,B 0,C 180,E1 -21765.482,E2 -21765.482} C_VEL
LIN {X 0,Y 193.671,Z 367.801,A -85,B 0,C 180,E1 -21769.546,E2 -21769.546} C_VEL
LIN {X 0,Y 191.972,Z 364.735,A -85,B 0,C 180,E1 -21773.695,E2 -21773.695} C_VEL
LIN {X 0,Y 190.837,Z 360.23,A -85,B 0,C 180,E1 -21777.89,E2 -21777.89} C_VEL
LIN {X 0,Y 190.655,Z 355.809,A -85,B 0,C 180,E1 -21781.056,E2 -21781.056} C_VEL
LIN {X 0,Y 190.695,Z 349.357,A -85,B 0,C 180,E1 -21784.74,E2 -21784.74} C_VEL
LIN {X 0,Y 191.072,Z 342.431,A -85,B 0,C 180,E1 -21787.928,E2 -21787.928} C_VEL
LIN {X 0,Y 191.679,Z 334.018,A -85,B 0,C 180,E1 -21791.099,E2 -21791.099} C_VEL
LIN {X 0,Y 192.644,Z 323.805,A -85,B 0,C 180,E1 -21794.256,E2 -21794.256} C_VEL
LIN {X 0,Y 193.805,Z 313.489,A -85,B 0,C 180,E1 -21796.865,E2 -21796.865} C_VEL
LIN {X 0,Y 195.075,Z 300.853,A -85,B 0,C 180,E1 -21799.467,E2 -21799.467} C_VEL
LIN {X 0,Y 195.872,Z 293.949,A -85,B 0,C 180,E1 -21800.649,E2 -21800.649} C_VEL
LIN {X 0,Y 193.845,Z 281.32,A -85,B 0,C 180,E1 -21802.512,E2 -21802.512} C_VEL
LIN {X 0,Y 191.741,Z 268.466,A -85,B 0,C 180,E1 -21804.036,E2 -21804.036} C_VEL
LIN {X 0,Y 191.216,Z 264.668,A -85,B 0,C 180,E1 -21804.445,E2 -21804.445} C_VEL
LIN {X 0,Y 191.569,Z 264.621,A -85,B 0,C 180,E1 -21808.485,E2 -21808.485} C_VEL
LIN {X 0,Y 192.088,Z 264.556,A -85,B 0,C 180,E1 -21813.286,E2 -21813.286} C_VEL
LIN {X 0,Y 192.387,Z 264.519,A -85,B 0,C 180,E1 -21816.517,E2 -21816.517} C_VEL
LIN {X 0,Y 192.505,Z 264.503,A -85,B 0,C 180,E1 -21821.083,E2 -21821.083} C_VEL
LIN {X 0,Y 192.491,Z 264.507,A -85,B 0,C 180,E1 -21826.075,E2 -21826.075} C_VEL
LIN {X 0,Y 192.51,Z 264.506,A -85,B 0,C 180,E1 -21830.055,E2 -21830.055} C_VEL
LIN {X 0,Y 192.56,Z 264.497,A -85,B 0,C 180,E1 -21834.27,E2 -21834.27} C_VEL
LIN {X 0,Y 192.608,Z 264.493,A -85,B 0,C 180,E1 -21837.061,E2 -21837.061} C_VEL
LIN {X 0,Y 192.624,Z 264.49,A -85,B 0,C 180,E1 -21841.685,E2 -21841.685} C_VEL
LIN {X 0,Y 192.683,Z 264.484,A -85,B 0,C 180,E1 -21846.345,E2 -21846.345} C_VEL
LIN {X 0,Y 192.735,Z 264.473,A -85,B 0,C 180,E1 -21851.457,E2 -21851.457} C_VEL
LIN {X 0,Y 192.767,Z 264.472,A -85,B 0,C 180,E1 -21855.214,E2 -21855.214} C_VEL
LIN {X 0,Y 192.948,Z 264.452,A -85,B 0,C 180,E1 -21859.566,E2 -21859.566} C_VEL
LIN {X 0,Y 192.967,Z 264.45,A -85,B 0,C 180,E1 -21863.727,E2 -21863.727} C_VEL
LIN {X 0,Y 193.256,Z 264.619,A -85,B 0,C 180,E1 -21867.916,E2 -21867.916} C_VEL
LIN {X 0,Y 193.987,Z 268.592,A -85,B 0,C 180,E1 -21871.038,E2 -21871.038} C_VEL
LIN {X 0,Y 193.971,Z 272.762,A -85,B 0,C 180,E1 -21874.155,E2 -21874.155} C_VEL
LIN {X 0,Y 193.327,Z 280.012,A -85,B 0,C 180,E1 -21879.415,E2 -21879.415} C_VEL
LIN {X 0,Y 192.975,Z 283.487,A -85,B 0,C 180,E1 -21881.921,E2 -21881.921} C_VEL
LIN {X 0,Y 194.959,Z 293.563,A -85,B 0,C 180,E1 -21882.888,E2 -21882.888} C_VEL
LIN {X 0,Y 196.353,Z 302.534,A -85,B 0,C 180,E1 -21883.981,E2 -21883.981} C_VEL
LIN {X 0,Y 197.57,Z 312.41,A -85,B 0,C 180,E1 -21885.474,E2 -21885.474} C_VEL
LIN {X 0,Y 197.798,Z 317.601,A -85,B 0,C 180,E1 -21886.393,E2 -21886.393} C_VEL
LIN {X 0,Y 196.616,Z 325.708,A -85,B 0,C 180,E1 -21887.957,E2 -21887.957} C_VEL
LIN {X 0,Y 195.291,Z 333.761,A -85,B 0,C 180,E1 -21889.875,E2 -21889.875} C_VEL
LIN {X 0,Y 193.891,Z 342.081,A -85,B 0,C 180,E1 -21892.37,E2 -21892.37} C_VEL
LIN {X 0,Y 192.637,Z 349.125,A -85,B 0,C 180,E1 -21895.125,E2 -21895.125} C_VEL
LIN {X 0,Y 191.721,Z 354.36,A -85,B 0,C 180,E1 -21897.707,E2 -21897.707} C_VEL
LIN {X 0,Y 190.831,Z 359.55,A -85,B 0,C 180,E1 -21901.037,E2 -21901.037} C_VEL
LIN {X 0,Y 190.379,Z 362.437,A -85,B 0,C 180,E1 -21903.624,E2 -21903.624} C_VEL
LIN {X 0,Y 190.249,Z 364.496,A -85,B 0,C 180,E1 -21906.232,E2 -21906.232} C_VEL
LIN {X 0,Y 190.408,Z 365.859,A -85,B 0,C 180,E1 -21909.184,E2 -21909.184} C_VEL
LIN {X 0,Y 191.037,Z 366.183,A -85,B 0,C 180,E1 -21912.627,E2 -21912.627} C_VEL
LIN {X 0,Y 191.512,Z 365.984,A -85,B 0,C 180,E1 -21914.207,E2 -21914.207} C_VEL
LIN {X 0,Y 192.542,Z 364.873,A -85,B 0,C 180,E1 -21916.888,E2 -21916.888} C_VEL
LIN {X 0,Y 193.895,Z 362.893,A -85,B 0,C 180,E1 -21919.568,E2 -21919.568} C_VEL
LIN {X 0,Y 195.777,Z 359.718,A -85,B 0,C 180,E1 -21922.391,E2 -21922.391} C_VEL
LIN {X 0,Y 197.666,Z 355.966,A -85,B 0,C 180,E1 -21924.861,E2 -21924.861} C_VEL
LIN {X 0,Y 199.533,Z 352.013,A -85,B 0,C 180,E1 -21926.912,E2 -21926.912} C_VEL
LIN {X 0,Y 201.92,Z 346.7,A -85,B 0,C 180,E1 -21929.09,E2 -21929.09} C_VEL
LIN {X 0,Y 204.563,Z 340.083,A -85,B 0,C 180,E1 -21931.25,E2 -21931.25} C_VEL
LIN {X 0,Y 207.175,Z 332.65,A -85,B 0,C 180,E1 -21933.196,E2 -21933.196} C_VEL
LIN {X 0,Y 208.013,Z 329.492,A -85,B 0,C 180,E1 -21933.945,E2 -21933.945} C_VEL
LIN {X 0,Y 207.936,Z 321.116,A -85,B 0,C 180,E1 -21936.072,E2 -21936.072} C_VEL
LIN {X 0,Y 207.123,Z 313.727,A -85,B 0,C 180,E1 -21937.822,E2 -21937.822} C_VEL
LIN {X 0,Y 205.664,Z 306.333,A -85,B 0,C 180,E1 -21939.496,E2 -21939.496} C_VEL
LIN {X 0,Y 203.469,Z 298.523,A -85,B 0,C 180,E1 -21941.236,E2 -21941.236} C_VEL
LIN {X 0,Y 201.423,Z 293.203,A -85,B 0,C 180,E1 -21942.486,E2 -21942.486} C_VEL
LIN {X 0,Y 199.715,Z 289.823,A -85,B 0,C 180,E1 -21943.32,E2 -21943.32} C_VEL
LIN {X 0,Y 197.91,Z 286.303,A -85,B 0,C 180,E1 -21944.233,E2 -21944.233} C_VEL
LIN {X 0,Y 197.825,Z 285.919,A -85,B 0,C 180,E1 -21944.397,E2 -21944.397} C_VEL
LIN {X 0,Y 197.068,Z 280.91,A -85,B 0,C 180,E1 -21949.728,E2 -21949.728} C_VEL
LIN {X 0,Y 196.508,Z 277.41,A -85,B 0,C 180,E1 -21953.84,E2 -21953.84} C_VEL
LIN {X 0,Y 196.051,Z 274.256,A -85,B 0,C 180,E1 -21957.945,E2 -21957.945} C_VEL
LIN {X 0,Y 195.863,Z 272.823,A -85,B 0,C 180,E1 -21960,E2 -21960} C_VEL
LIN {X 0,Y 195.517,Z 271.56,A -85,B 0,C 180,E1 -21962.06,E2 -21962.06} C_VEL
LIN {X 0,Y 194.29,Z 268.646,A -85,B 0,C 180,E1 -21968.319,E2 -21968.319} C_VEL
LIN {X 0,Y 193.79,Z 267.336,A -85,B 0,C 180,E1 -21972.568,E2 -21972.568} C_VEL
LIN {X 0,Y 193.357,Z 266.615,A -85,B 0,C 180,E1 -21976.904,E2 -21976.904} C_VEL
LIN {X 0,Y 193.197,Z 266.528,A -85,B 0,C 180,E1 -21981.332,E2 -21981.332} C_VEL
LIN {X 0,Y 193.535,Z 267.218,A -85,B 0,C 180,E1 -21985.834,E2 -21985.834} C_VEL
LIN {X 0,Y 193.861,Z 267.704,A -85,B 0,C 180,E1 -21988.118,E2 -21988.118} C_VEL
LIN {X 0,Y 194.896,Z 270.517,A -85,B 0,C 180,E1 -21993.964,E2 -21993.964} C_VEL
LIN {X 0,Y 195.903,Z 273.325,A -85,B 0,C 180,E1 -21997.885,E2 -21997.885} C_VEL
LIN {X 0,Y 197.676,Z 277.637,A -85,B 0,C 180,E1 -22002.494,E2 -22002.494} C_VEL
LIN {X 0,Y 198.607,Z 280.725,A -85,B 0,C 180,E1 -22005.05,E2 -22005.05} C_VEL
LIN {X 0,Y 199.844,Z 286.962,A -85,B 0,C 180,E1 -22009.12,E2 -22009.12} C_VEL
LIN {X 0,Y 200.306,Z 290.922,A -85,B 0,C 180,E1 -22011.265,E2 -22011.265} C_VEL
LIN {X 0,Y 200.123,Z 295.942,A -85,B 0,C 180,E1 -22013.422,E2 -22013.422} C_VEL
LIN {X 0,Y 204.167,Z 308.958,A -85,B 0,C 180,E1 -22015.63,E2 -22015.63} C_VEL
LIN {X 0,Y 205.986,Z 318.111,A -85,B 0,C 180,E1 -22017.183,E2 -22017.183} C_VEL
LIN {X 0,Y 206.763,Z 326.449,A -85,B 0,C 180,E1 -22018.621,E2 -22018.621} C_VEL
LIN {X 0,Y 205.706,Z 335.724,A -85,B 0,C 180,E1 -22020.12,E2 -22020.12} C_VEL
LIN {X 0,Y 204.594,Z 344.154,A -85,B 0,C 180,E1 -22021.815,E2 -22021.815} C_VEL
LIN {X 0,Y 203.723,Z 348.635,A -85,B 0,C 180,E1 -22022.8,E2 -22022.8} C_VEL
LIN {X 0,Y 201.248,Z 356.216,A -85,B 0,C 180,E1 -22024.672,E2 -22024.672} C_VEL
LIN {X 0,Y 198.427,Z 363.913,A -85,B 0,C 180,E1 -22027.07,E2 -22027.07} C_VEL
LIN {X 0,Y 195.865,Z 371.287,A -85,B 0,C 180,E1 -22030.07,E2 -22030.07} C_VEL
LIN {X 0,Y 193.602,Z 376.817,A -85,B 0,C 180,E1 -22033.118,E2 -22033.118} C_VEL
LIN {X 0,Y 193.198,Z 377.751,A -85,B 0,C 180,E1 -22033.742,E2 -22033.742} C_VEL
LIN {X 0,Y 191.652,Z 379.988,A -85,B 0,C 180,E1 -22035.314,E2 -22035.314} C_VEL
LIN {X 0,Y 189.389,Z 381.837,A -85,B 0,C 180,E1 -22036.876,E2 -22036.876} C_VEL
LIN {X 0,Y 184.796,Z 384.397,A -85,B 0,C 180,E1 -22040.154,E2 -22040.154} C_VEL
LIN {X 0,Y 183.42,Z 385.351,A -85,B 0,C 180,E1 -22042.239,E2 -22042.239} C_VEL
LIN {X 0,Y 183.373,Z 385.32,A -85,B 0,C 180,E1 -22042.545,E2 -22042.545} C_VEL
LIN {X 0,Y 183.308,Z 385.843,A -85,B 0,C 180,E1 -22045.603,E2 -22045.603} C_VEL
LIN {X 0,Y 183.518,Z 385.614,A -85,B 0,C 180,E1 -22047.806,E2 -22047.806} C_VEL
LIN {X 0,Y 183.64,Z 384.782,A -85,B 0,C 180,E1 -22050,E2 -22050} C_VEL
LIN {X 0,Y 183.671,Z 383.407,A -85,B 0,C 180,E1 -22052.193,E2 -22052.193} C_VEL
LIN {X 0,Y 183.961,Z 379.891,A -85,B 0,C 180,E1 -22056.078,E2 -22056.078} C_VEL
LIN {X 0,Y 184.282,Z 382.644,A -85,B 0,C 180,E1 -22060.993,E2 -22060.993} C_VEL
LIN {X 0,Y 185.721,Z 383.78,A -85,B 0,C 180,E1 -22065.361,E2 -22065.361} C_VEL
LIN {X 0,Y 188.697,Z 383.75,A -85,B 0,C 180,E1 -22069.585,E2 -22069.585} C_VEL
LIN {X 0,Y 192.824,Z 382.511,A -85,B 0,C 180,E1 -22073.636,E2 -22073.636} C_VEL
LIN {X 0,Y 198.036,Z 380.099,A -85,B 0,C 180,E1 -22077.475,E2 -22077.475} C_VEL
LIN {X 0,Y 201.077,Z 378.458,A -85,B 0,C 180,E1 -22079.297,E2 -22079.297} C_VEL
LIN {X 0,Y 208.263,Z 374.237,A -85,B 0,C 180,E1 -22082.68,E2 -22082.68} C_VEL
LIN {X 0,Y 216.369,Z 368.759,A -85,B 0,C 180,E1 -22085.78,E2 -22085.78} C_VEL
LIN {X 0,Y 220.516,Z 365.591,A -85,B 0,C 180,E1 -22087.269,E2 -22087.269} C_VEL
LIN {X 0,Y 224.748,Z 361.214,A -85,B 0,C 180,E1 -22089.871,E2 -22089.871} C_VEL
LIN {X 0,Y 227.894,Z 357.601,A -85,B 0,C 180,E1 -22092.257,E2 -22092.257} C_VEL
LIN {X 0,Y 228.29,Z 357.11,A -85,B 0,C 180,E1 -22092.632,E2 -22092.632} C_VEL
LIN {X 0,Y 229.529,Z 355.133,A -85,B 0,C 180,E1 -22094.769,E2 -22094.769} C_VEL
LIN {X 0,Y 230.032,Z 353.881,A -85,B 0,C 180,E1 -22097.767,E2 -22097.767} C_VEL
LIN {X 0,Y 230.053,Z 353.737,A -85,B 0,C 180,E1 -22100.093,E2 -22100.093} C_VEL
LIN {X 0,Y 229.37,Z 354.58,A -85,B 0,C 180,E1 -22102.812,E2 -22102.812} C_VEL
LIN {X 0,Y 228.712,Z 355.42,A -85,B 0,C 180,E1 -22104.279,E2 -22104.279} C_VEL
LIN {X 0,Y 226.877,Z 356.764,A -85,B 0,C 180,E1 -22105.035,E2 -22105.035} C_VEL
LIN {X 0,Y 218.213,Z 362.173,A -85,B 0,C 180,E1 -22107.899,E2 -22107.899} C_VEL
LIN {X 0,Y 212.306,Z 365.288,A -85,B 0,C 180,E1 -22110.228,E2 -22110.228} C_VEL
LIN {X 0,Y 205.074,Z 368.328,A -85,B 0,C 180,E1 -22113.544,E2 -22113.544} C_VEL
LIN {X 0,Y 198.876,Z 370.081,A -85,B 0,C 180,E1 -22117.125,E2 -22117.125} C_VEL
LIN {X 0,Y 193.632,Z 370.559,A -85,B 0,C 180,E1 -22120.934,E2 -22120.934} C_VEL
LIN {X 0,Y 189.389,Z 369.76,A -85,B 0,C 180,E1 -22124.944,E2 -22124.944} C_VEL
LIN {X 0,Y 186.691,Z 367.681,A -85,B 0,C 180,E1 -22129.151,E2 -22129.151} C_VEL
LIN {X 0,Y 184.944,Z 364.312,A -85,B 0,C 180,E1 -22133.454,E2 -22133.454} C_VEL
LIN {X 0,Y 183.779,Z 359.439,A -85,B 0,C 180,E1 -22137.809,E2 -22137.809} C_VEL
LIN {X 0,Y 183.62,Z 354.754,A -85,B 0,C 180,E1 -22141.097,E2 -22141.097} C_VEL
LIN {X 0,Y 183.688,Z 348.198,A -85,B 0,C 180,E1 -22144.788,E2 -22144.788} C_VEL
LIN {X 0,Y 184.119,Z 340.264,A -85,B 0,C 180,E1 -22148.391,E2 -22148.391} C_VEL
LIN {X 0,Y 184.74,Z 331.87,A -85,B 0,C 180,E1 -22151.521,E2 -22151.521} C_VEL
LIN {X 0,Y 185.841,Z 321.114,A -85,B 0,C 180,E1 -22154.79,E2 -22154.79} C_VEL
LIN {X 0,Y 186.912,Z 310.208,A -85,B 0,C 180,E1 -22157.506,E2 -22157.506} C_VEL
LIN {X 0,Y 188.399,Z 297.28,A -85,B 0,C 180,E1 -22160.088,E2 -22160.088} C_VEL
LIN {X 0,Y 188.677,Z 293.237,A -85,B 0,C 180,E1 -22160.78,E2 -22160.78} C_VEL
LIN {X 0,Y 186.606,Z 281.037,A -85,B 0,C 180,E1 -22162.626,E2 -22162.626} C_VEL
LIN {X 0,Y 184.49,Z 267.665,A -85,B 0,C 180,E1 -22164.238,E2 -22164.238} C_VEL
LIN {X 0,Y 184.188,Z 265.543,A -85,B 0,C 180,E1 -22164.481,E2 -22164.481} C_VEL
LIN {X 0,Y 184.637,Z 265.486,A -85,B 0,C 180,E1 -22169.659,E2 -22169.659} C_VEL
LIN {X 0,Y 185.044,Z 265.433,A -85,B 0,C 180,E1 -22173.324,E2 -22173.324} C_VEL
LIN {X 0,Y 185.363,Z 265.397,A -85,B 0,C 180,E1 -22177.347,E2 -22177.347} C_VEL
LIN {X 0,Y 185.459,Z 265.381,A -85,B 0,C 180,E1 -22180.719,E2 -22180.719} C_VEL
LIN {X 0,Y 185.46,Z 265.383,A -85,B 0,C 180,E1 -22186.056,E2 -22186.056} C_VEL
LIN {X 0,Y 185.46,Z 265.384,A -85,B 0,C 180,E1 -22189.893,E2 -22189.893} C_VEL
LIN {X 0,Y 185.503,Z 265.377,A -85,B 0,C 180,E1 -22192.714,E2 -22192.714} C_VEL
LIN {X 0,Y 185.534,Z 265.373,A -85,B 0,C 180,E1 -22197.972,E2 -22197.972} C_VEL
LIN {X 0,Y 185.55,Z 265.374,A -85,B 0,C 180,E1 -22200.595,E2 -22200.595} C_VEL
LIN {X 0,Y 185.583,Z 265.367,A -85,B 0,C 180,E1 -22205.381,E2 -22205.381} C_VEL
LIN {X 0,Y 185.678,Z 265.352,A -85,B 0,C 180,E1 -22211.133,E2 -22211.133} C_VEL
LIN {X 0,Y 185.699,Z 265.354,A -85,B 0,C 180,E1 -22214.637,E2 -22214.637} C_VEL
LIN {X 0,Y 185.891,Z 265.331,A -85,B 0,C 180,E1 -22219.419,E2 -22219.419} C_VEL
LIN {X 0,Y 185.932,Z 265.327,A -85,B 0,C 180,E1 -22223.488,E2 -22223.488} C_VEL
LIN {X 0,Y 186.074,Z 265.408,A -85,B 0,C 180,E1 -22227.158,E2 -22227.158} C_VEL
LIN {X 0,Y 186.968,Z 268.828,A -85,B 0,C 180,E1 -22230,E2 -22230} C_VEL
LIN {X 0,Y 187.064,Z 273.003,A -85,B 0,C 180,E1 -22233.23,E2 -22233.23} C_VEL
LIN {X 0,Y 186.522,Z 278.829,A -85,B 0,C 180,E1 -22237.578,E2 -22237.578} C_VEL
LIN {X 0,Y 186.045,Z 283.767,A -85,B 0,C 180,E1 -22241.232,E2 -22241.232} C_VEL
LIN {X 0,Y 188.164,Z 294.6,A -85,B 0,C 180,E1 -22242.333,E2 -22242.333} C_VEL
LIN {X 0,Y 189.499,Z 303.487,A -85,B 0,C 180,E1 -22243.471,E2 -22243.471} C_VEL
LIN {X 0,Y 190.637,Z 312.847,A -85,B 0,C 180,E1 -22244.955,E2 -22244.955} C_VEL
LIN {X 0,Y 190.886,Z 318.178,A -85,B 0,C 180,E1 -22245.94,E2 -22245.94} C_VEL
LIN {X 0,Y 189.668,Z 326.095,A -85,B 0,C 180,E1 -22247.521,E2 -22247.521} C_VEL
LIN {X 0,Y 188.253,Z 334.613,A -85,B 0,C 180,E1 -22249.633,E2 -22249.633} C_VEL
LIN {X 0,Y 186.861,Z 342.465,A -85,B 0,C 180,E1 -22252.093,E2 -22252.093} C_VEL
LIN {X 0,Y 185.673,Z 348.991,A -85,B 0,C 180,E1 -22254.709,E2 -22254.709} C_VEL
LIN {X 0,Y 184.734,Z 353.929,A -85,B 0,C 180,E1 -22257.163,E2 -22257.163} C_VEL
LIN {X 0,Y 183.996,Z 358.108,A -85,B 0,C 180,E1 -22259.772,E2 -22259.772} C_VEL
LIN {X 0,Y 183.433,Z 361.535,A -85,B 0,C 180,E1 -22262.551,E2 -22262.551} C_VEL
LIN {X 0,Y 183.176,Z 363.879,A -85,B 0,C 180,E1 -22265.135,E2 -22265.135} C_VEL
LIN {X 0,Y 183.213,Z 365.55,A -85,B 0,C 180,E1 -22267.861,E2 -22267.861} C_VEL
LIN {X 0,Y 183.508,Z 366.449,A -85,B 0,C 180,E1 -22270.622,E2 -22270.622} C_VEL
LIN {X 0,Y 184.179,Z 366.547,A -85,B 0,C 180,E1 -22273.529,E2 -22273.529} C_VEL
LIN {X 0,Y 185.473,Z 365.543,A -85,B 0,C 180,E1 -22276.994,E2 -22276.994} C_VEL
LIN {X 0,Y 187.195,Z 363.299,A -85,B 0,C 180,E1 -22280.338,E2 -22280.338} C_VEL
LIN {X 0,Y 189.494,Z 359.645,A -85,B 0,C 180,E1 -22283.6,E2 -22283.6} C_VEL
LIN {X 0,Y 192.085,Z 354.767,A -85,B 0,C 180,E1 -22286.714,E2 -22286.714} C_VEL
LIN {X 0,Y 195.349,Z 348.192,A -85,B 0,C 180,E1 -22289.756,E2 -22289.756} C_VEL
LIN {X 0,Y 198.485,Z 340.82,A -85,B 0,C 180,E1 -22292.277,E2 -22292.277} C_VEL
LIN {X 0,Y 201.147,Z 333.685,A -85,B 0,C 180,E1 -22294.208,E2 -22294.208} C_VEL
LIN {X 0,Y 201.901,Z 331.239,A -85,B 0,C 180,E1 -22294.829,E2 -22294.829} C_VEL
LIN {X 0,Y 201.924,Z 322.375,A -85,B 0,C 180,E1 -22297.219,E2 -22297.219} C_VEL
LIN {X 0,Y 201.174,Z 314.728,A -85,B 0,C 180,E1 -22299.151,E2 -22299.151} C_VEL
LIN {X 0,Y 199.627,Z 306.758,A -85,B 0,C 180,E1 -22301.095,E2 -22301.095} C_VEL
LIN {X 0,Y 197.135,Z 298.394,A -85,B 0,C 180,E1 -22303.137,E2 -22303.137} C_VEL
LIN {X 0,Y 195.32,Z 294.46,A -85,B 0,C 180,E1 -22304.268,E2 -22304.268} C_VEL
LIN {X 0,Y 193.233,Z 290.635,A -85,B 0,C 180,E1 -22305.385,E2 -22305.385} C_VEL
LIN {X 0,Y 191.043,Z 286.855,A -85,B 0,C 180,E1 -22306.572,E2 -22306.572} C_VEL
LIN {X 0,Y 190.922,Z 286.482,A -85,B 0,C 180,E1 -22306.699,E2 -22306.699} C_VEL
LIN {X 0,Y 190.389,Z 282.298,A -85,B 0,C 180,E1 -22311.509,E2 -22311.509} C_VEL
LIN {X 0,Y 189.849,Z 279.05,A -85,B 0,C 180,E1 -22315.754,E2 -22315.754} C_VEL
LIN {X 0,Y 189.567,Z 276.099,A -85,B 0,C 180,E1 -22320,E2 -22320} C_VEL
LIN {X 0,Y 189.244,Z 274.867,A -85,B 0,C 180,E1 -22322.128,E2 -22322.128} C_VEL
LIN {X 0,Y 188.122,Z 272.139,A -85,B 0,C 180,E1 -22328.594,E2 -22328.594} C_VEL
LIN {X 0,Y 187.646,Z 270.895,A -85,B 0,C 180,E1 -22333.147,E2 -22333.147} C_VEL
LIN {X 0,Y 187.299,Z 270.365,A -85,B 0,C 180,E1 -22337.468,E2 -22337.468} C_VEL
LIN {X 0,Y 187.315,Z 270.534,A -85,B 0,C 180,E1 -22342.036,E2 -22342.036} C_VEL
LIN {X 0,Y 187.782,Z 271.418,A -85,B 0,C 180,E1 -22346.687,E2 -22346.687} C_VEL
LIN {X 0,Y 188.09,Z 272.156,A -85,B 0,C 180,E1 -22349.061,E2 -22349.061} C_VEL
LIN {X 0,Y 189.068,Z 274.551,A -85,B 0,C 180,E1 -22353.888,E2 -22353.888} C_VEL
LIN {X 0,Y 190.519,Z 278.586,A -85,B 0,C 180,E1 -22359.226,E2 -22359.226} C_VEL
LIN {X 0,Y 191.978,Z 282.203,A -85,B 0,C 180,E1 -22362.932,E2 -22362.932} C_VEL
LIN {X 0,Y 193.023,Z 286.481,A -85,B 0,C 180,E1 -22366.228,E2 -22366.228} C_VEL
LIN {X 0,Y 194.001,Z 291.65,A -85,B 0,C 180,E1 -22369.531,E2 -22369.531} C_VEL
LIN {X 0,Y 194.115,Z 295.649,A -85,B 0,C 180,E1 -22371.487,E2 -22371.487} C_VEL
LIN {X 0,Y 198.062,Z 308.061,A -85,B 0,C 180,E1 -22373.817,E2 -22373.817} C_VEL
LIN {X 0,Y 200.207,Z 318.841,A -85,B 0,C 180,E1 -22375.83,E2 -22375.83} C_VEL
LIN {X 0,Y 200.966,Z 326.821,A -85,B 0,C 180,E1 -22377.321,E2 -22377.321} C_VEL
LIN {X 0,Y 199.983,Z 335.373,A -85,B 0,C 180,E1 -22378.79,E2 -22378.79} C_VEL
LIN {X 0,Y 198.629,Z 344.08,A -85,B 0,C 180,E1 -22380.598,E2 -22380.598} C_VEL
LIN {X 0,Y 197.497,Z 349.461,A -85,B 0,C 180,E1 -22381.868,E2 -22381.868} C_VEL
LIN {X 0,Y 194.895,Z 356.846,A -85,B 0,C 180,E1 -22383.785,E2 -22383.785} C_VEL
LIN {X 0,Y 192.508,Z 362.984,A -85,B 0,C 180,E1 -22385.751,E2 -22385.751} C_VEL
LIN {X 0,Y 190.594,Z 367.9,A -85,B 0,C 180,E1 -22387.682,E2 -22387.682} C_VEL
LIN {X 0,Y 188.335,Z 373.408,A -85,B 0,C 180,E1 -22390.376,E2 -22390.376} C_VEL
LIN {X 0,Y 186.263,Z 378.04,A -85,B 0,C 180,E1 -22393.306,E2 -22393.306} C_VEL
LIN {X 0,Y 184.611,Z 382.008,A -85,B 0,C 180,E1 -22396.796,E2 -22396.796} C_VEL
LIN {X 0,Y 183.948,Z 383.718,A -85,B 0,C 180,E1 -22398.987,E2 -22398.987} C_VEL
LIN {X 0,Y 183.373,Z 385.32,A -85,B 0,C 180,E1 -22402.545,E2 -22402.545} C_VEL
LIN {X 0,Y 182.651,Z 385.765,A -85,B 0,C 180,E1 -22404.378,E2 -22404.378} C_VEL
LIN {X 0,Y 181.145,Z 385.727,A -85,B 0,C 180,E1 -22406.19,E2 -22406.19} C_VEL
LIN {X 0,Y 177.696,Z 384.423,A -85,B 0,C 180,E1 -22409.844,E2 -22409.844} C_VEL
LIN {X 0,Y 176.604,Z 382.741,A -85,B 0,C 180,E1 -22412.351,E2 -22412.351} C_VEL
LIN {X 0,Y 176.948,Z 378.988,A -85,B 0,C 180,E1 -22416.247,E2 -22416.247} C_VEL
LIN {X 0,Y 177.038,Z 378.662,A -85,B 0,C 180,E1 -22416.617,E2 -22416.617} C_VEL
LIN {X 0,Y 177.364,Z 381.517,A -85,B 0,C 180,E1 -22421.428,E2 -22421.428} C_VEL
LIN {X 0,Y 178.919,Z 382.938,A -85,B 0,C 180,E1 -22425.96,E2 -22425.96} C_VEL
LIN {X 0,Y 182.031,Z 383.223,A -85,B 0,C 180,E1 -22430.334,E2 -22430.334} C_VEL
LIN {X 0,Y 186.332,Z 382.342,A -85,B 0,C 180,E1 -22434.513,E2 -22434.513} C_VEL
LIN {X 0,Y 191.776,Z 380.323,A -85,B 0,C 180,E1 -22438.452,E2 -22438.452} C_VEL
LIN {X 0,Y 194.928,Z 378.899,A -85,B 0,C 180,E1 -22440.316,E2 -22440.316} C_VEL
LIN {X 0,Y 202.387,Z 375.141,A -85,B 0,C 180,E1 -22443.753,E2 -22443.753} C_VEL
LIN {X 0,Y 210.748,Z 370.185,A -85,B 0,C 180,E1 -22446.889,E2 -22446.889} C_VEL
LIN {X 0,Y 215.047,Z 367.287,A -85,B 0,C 180,E1 -22448.386,E2 -22448.386} C_VEL
LIN {X 0,Y 219.448,Z 363.304,A -85,B 0,C 180,E1 -22451.036,E2 -22451.036} C_VEL
LIN {X 0,Y 220.791,Z 361.987,A -85,B 0,C 180,E1 -22451.948,E2 -22451.948} C_VEL
LIN {X 0,Y 222.503,Z 360.226,A -85,B 0,C 180,E1 -22453.408,E2 -22453.408} C_VEL
LIN {X 0,Y 223.8,Z 358.264,A -85,B 0,C 180,E1 -22456.301,E2 -22456.301} C_VEL
LIN {X 0,Y 224.047,Z 357.627,A -85,B 0,C 180,E1 -22458.838,E2 -22458.838} C_VEL
LIN {X 0,Y 223.55,Z 357.939,A -85,B 0,C 180,E1 -22461.81,E2 -22461.81} C_VEL
LIN {X 0,Y 222.996,Z 358.466,A -85,B 0,C 180,E1 -22463.215,E2 -22463.215} C_VEL
LIN {X 0,Y 221.41,Z 359.515,A -85,B 0,C 180,E1 -22464.04,E2 -22464.04} C_VEL
LIN {X 0,Y 212.455,Z 364.367,A -85,B 0,C 180,E1 -22466.919,E2 -22466.919} C_VEL
LIN {X 0,Y 206.343,Z 367.123,A -85,B 0,C 180,E1 -22469.276,E2 -22469.276} C_VEL
LIN {X 0,Y 198.862,Z 369.681,A -85,B 0,C 180,E1 -22472.65,E2 -22472.65} C_VEL
LIN {X 0,Y 192.405,Z 370.992,A -85,B 0,C 180,E1 -22476.31,E2 -22476.31} C_VEL
LIN {X 0,Y 186.982,Z 371.083,A -85,B 0,C 180,E1 -22480.228,E2 -22480.228} C_VEL
LIN {X 0,Y 182.545,Z 369.922,A -85,B 0,C 180,E1 -22484.366,E2 -22484.366} C_VEL
LIN {X 0,Y 179.723,Z 367.47,A -85,B 0,C 180,E1 -22488.725,E2 -22488.725} C_VEL
LIN {X 0,Y 177.921,Z 363.73,A -85,B 0,C 180,E1 -22493.195,E2 -22493.195} C_VEL
LIN {X 0,Y 176.732,Z 358.535,A -85,B 0,C 180,E1 -22497.721,E2 -22497.721} C_VEL
LIN {X 0,Y 176.605,Z 353.549,A -85,B 0,C 180,E1 -22501.14,E2 -22501.14} C_VEL
LIN {X 0,Y 176.675,Z 347.47,A -85,B 0,C 180,E1 -22504.563,E2 -22504.563} C_VEL
LIN {X 0,Y 177.046,Z 340.114,A -85,B 0,C 180,E1 -22507.987,E2 -22507.987} C_VEL
LIN {X 0,Y 177.705,Z 331.128,A -85,B 0,C 180,E1 -22511.405,E2 -22511.405} C_VEL
LIN {X 0,Y 178.796,Z 320.256,A -85,B 0,C 180,E1 -22514.803,E2 -22514.803} C_VEL
LIN {X 0,Y 179.899,Z 309.059,A -85,B 0,C 180,E1 -22517.624,E2 -22517.624} C_VEL
LIN {X 0,Y 181.287,Z 296.916,A -85,B 0,C 180,E1 -22520.125,E2 -22520.125} C_VEL
LIN {X 0,Y 181.58,Z 293.994,A -85,B 0,C 180,E1 -22520.643,E2 -22520.643} C_VEL
LIN {X 0,Y 179.364,Z 280.896,A -85,B 0,C 180,E1 -22522.697,E2 -22522.697} C_VEL
LIN {X 0,Y 177.159,Z 266.419,A -85,B 0,C 180,E1 -22524.534,E2 -22524.534} C_VEL
LIN {X 0,Y 177.566,Z 266.365,A -85,B 0,C 180,E1 -22529.453,E2 -22529.453} C_VEL
LIN {X 0,Y 178.035,Z 266.303,A -85,B 0,C 180,E1 -22534.005,E2 -22534.005} C_VEL
LIN {X 0,Y 178.344,Z 266.271,A -85,B 0,C 180,E1 -22539.088,E2 -22539.088} C_VEL
LIN {X 0,Y 178.395,Z 266.261,A -85,B 0,C 180,E1 -22542.047,E2 -22542.047} C_VEL
LIN {X 0,Y 178.395,Z 266.265,A -85,B 0,C 180,E1 -22545.164,E2 -22545.164} C_VEL
LIN {X 0,Y 178.401,Z 266.261,A -85,B 0,C 180,E1 -22548.461,E2 -22548.461} C_VEL
LIN {X 0,Y 178.421,Z 266.258,A -85,B 0,C 180,E1 -22553.782,E2 -22553.782} C_VEL
LIN {X 0,Y 178.486,Z 266.255,A -85,B 0,C 180,E1 -22556.546,E2 -22556.546} C_VEL
LIN {X 0,Y 178.447,Z 266.256,A -85,B 0,C 180,E1 -22561.795,E2 -22561.795} C_VEL
LIN {X 0,Y 178.518,Z 266.248,A -85,B 0,C 180,E1 -22564.889,E2 -22564.889} C_VEL
LIN {X 0,Y 178.625,Z 266.231,A -85,B 0,C 180,E1 -22570.784,E2 -22570.784} C_VEL
LIN {X 0,Y 178.662,Z 266.228,A -85,B 0,C 180,E1 -22576.348,E2 -22576.348} C_VEL
LIN {X 0,Y 178.908,Z 266.202,A -85,B 0,C 180,E1 -22580.959,E2 -22580.959} C_VEL
LIN {X 0,Y 178.933,Z 266.32,A -85,B 0,C 180,E1 -22586.481,E2 -22586.481} C_VEL
LIN {X 0,Y 180.042,Z 270.434,A -85,B 0,C 180,E1 -22590,E2 -22590} C_VEL
LIN {X 0,Y 180.085,Z 274.684,A -85,B 0,C 180,E1 -22593.356,E2 -22593.356} C_VEL
LIN {X 0,Y 179.471,Z 280.584,A -85,B 0,C 180,E1 -22597.877,E2 -22597.877} C_VEL
LIN {X 0,Y 179.098,Z 284.079,A -85,B 0,C 180,E1 -22600.522,E2 -22600.522} C_VEL
LIN {X 0,Y 181.26,Z 295.151,A -85,B 0,C 180,E1 -22601.703,E2 -22601.703} C_VEL
LIN {X 0,Y 182.524,Z 303.319,A -85,B 0,C 180,E1 -22602.791,E2 -22602.791} C_VEL
LIN {X 0,Y 183.643,Z 312.951,A -85,B 0,C 180,E1 -22604.356,E2 -22604.356} C_VEL
LIN {X 0,Y 184.052,Z 317.903,A -85,B 0,C 180,E1 -22605.306,E2 -22605.306} C_VEL
LIN {X 0,Y 182.865,Z 325.739,A -85,B 0,C 180,E1 -22606.905,E2 -22606.905} C_VEL
LIN {X 0,Y 181.464,Z 333.773,A -85,B 0,C 180,E1 -22608.926,E2 -22608.926} C_VEL
LIN {X 0,Y 179.881,Z 342.566,A -85,B 0,C 180,E1 -22611.712,E2 -22611.712} C_VEL
LIN {X 0,Y 178.663,Z 349.013,A -85,B 0,C 180,E1 -22614.366,E2 -22614.366} C_VEL
LIN {X 0,Y 177.649,Z 354.261,A -85,B 0,C 180,E1 -22617.062,E2 -22617.062} C_VEL
LIN {X 0,Y 176.815,Z 358.847,A -85,B 0,C 180,E1 -22620.067,E2 -22620.067} C_VEL
LIN {X 0,Y 176.244,Z 362.374,A -85,B 0,C 180,E1 -22623.132,E2 -22623.132} C_VEL
LIN {X 0,Y 176.076,Z 365.41,A -85,B 0,C 180,E1 -22627.032,E2 -22627.032} C_VEL
LIN {X 0,Y 176.439,Z 366.802,A -85,B 0,C 180,E1 -22630.815,E2 -22630.815} C_VEL
LIN {X 0,Y 176.818,Z 367.08,A -85,B 0,C 180,E1 -22632.508,E2 -22632.508} C_VEL
LIN {X 0,Y 177.676,Z 366.799,A -85,B 0,C 180,E1 -22635.397,E2 -22635.397} C_VEL
LIN {X 0,Y 178.934,Z 365.704,A -85,B 0,C 180,E1 -22638.268,E2 -22638.268} C_VEL
LIN {X 0,Y 180.751,Z 363.376,A -85,B 0,C 180,E1 -22641.529,E2 -22641.529} C_VEL
LIN {X 0,Y 183.289,Z 359.624,A -85,B 0,C 180,E1 -22644.889,E2 -22644.889} C_VEL
LIN {X 0,Y 186.14,Z 354.628,A -85,B 0,C 180,E1 -22648.089,E2 -22648.089} C_VEL
LIN {X 0,Y 189.637,Z 347.802,A -85,B 0,C 180,E1 -22651.198,E2 -22651.198} C_VEL
LIN {X 0,Y 192.552,Z 341.409,A -85,B 0,C 180,E1 -22653.41,E2 -22653.41} C_VEL
LIN {X 0,Y 195.239,Z 334.619,A -85,B 0,C 180,E1 -22655.304,E2 -22655.304} C_VEL
LIN {X 0,Y 195.777,Z 332.729,A -85,B 0,C 180,E1 -22655.819,E2 -22655.819} C_VEL
LIN {X 0,Y 196.014,Z 323.525,A -85,B 0,C 180,E1 -22658.493,E2 -22658.493} C_VEL
LIN {X 0,Y 195.35,Z 315.833,A -85,B 0,C 180,E1 -22660.562,E2 -22660.562} C_VEL
LIN {X 0,Y 193.909,Z 308.11,A -85,B 0,C 180,E1 -22662.601,E2 -22662.601} C_VEL
LIN {X 0,Y 191.55,Z 300.465,A -85,B 0,C 180,E1 -22664.709,E2 -22664.709} C_VEL
LIN {X 0,Y 189.032,Z 295.521,A -85,B 0,C 180,E1 -22666.358,E2 -22666.358} C_VEL
LIN {X 0,Y 186.835,Z 291.667,A -85,B 0,C 180,E1 -22667.692,E2 -22667.692} C_VEL
LIN {X 0,Y 184.583,Z 288.226,A -85,B 0,C 180,E1 -22669.025,E2 -22669.025} C_VEL
LIN {X 0,Y 184.104,Z 287.011,A -85,B 0,C 180,E1 -22669.414,E2 -22669.414} C_VEL
LIN {X 0,Y 183.605,Z 283.17,A -85,B 0,C 180,E1 -22674.396,E2 -22674.396} C_VEL
LIN {X 0,Y 183.374,Z 280.807,A -85,B 0,C 180,E1 -22677.803,E2 -22677.803} C_VEL
LIN {X 0,Y 183.259,Z 279.413,A -85,B 0,C 180,E1 -22680,E2 -22680} C_VEL
LIN {X 0,Y 182.899,Z 278.12,A -85,B 0,C 180,E1 -22682.475,E2 -22682.475} C_VEL
LIN {X 0,Y 181.974,Z 275.636,A -85,B 0,C 180,E1 -22688.887,E2 -22688.887} C_VEL
LIN {X 0,Y 181.579,Z 274.605,A -85,B 0,C 180,E1 -22693.428,E2 -22693.428} C_VEL
LIN {X 0,Y 181.329,Z 274.25,A -85,B 0,C 180,E1 -22698.063,E2 -22698.063} C_VEL
LIN {X 0,Y 181.452,Z 274.575,A -85,B 0,C 180,E1 -22702.788,E2 -22702.788} C_VEL
LIN {X 0,Y 181.997,Z 275.706,A -85,B 0,C 180,E1 -22707.606,E2 -22707.606} C_VEL
LIN {X 0,Y 182.845,Z 277.926,A -85,B 0,C 180,E1 -22712.555,E2 -22712.555} C_VEL
LIN {X 0,Y 183.867,Z 280.565,A -85,B 0,C 180,E1 -22716.612,E2 -22716.612} C_VEL
LIN {X 0,Y 185.549,Z 284.789,A -85,B 0,C 180,E1 -22721.516,E2 -22721.516} C_VEL
LIN {X 0,Y 186.543,Z 287.906,A -85,B 0,C 180,E1 -22724.289,E2 -22724.289} C_VEL
LIN {X 0,Y 187.678,Z 293.978,A -85,B 0,C 180,E1 -22728.499,E2 -22728.499} C_VEL
LIN {X 0,Y 187.934,Z 295.187,A -85,B 0,C 180,E1 -22729.194,E2 -22729.194} C_VEL
LIN {X 0,Y 190.227,Z 301.16,A -85,B 0,C 180,E1 -22730.583,E2 -22730.583} C_VEL
LIN {X 0,Y 193.05,Z 311.28,A -85,B 0,C 180,E1 -22732.689,E2 -22732.689} C_VEL
LIN {X 0,Y 194.547,Z 319.609,A -85,B 0,C 180,E1 -22734.373,E2 -22734.373} C_VEL
LIN {X 0,Y 195.166,Z 327.238,A -85,B 0,C 180,E1 -22735.918,E2 -22735.918} C_VEL
LIN {X 0,Y 195.11,Z 331.089,A -85,B 0,C 180,E1 -22736.663,E2 -22736.663} C_VEL
LIN {X 0,Y 193.204,Z 341.861,A -85,B 0,C 180,E1 -22738.778,E2 -22738.778} C_VEL
LIN {X 0,Y 191.907,Z 348.428,A -85,B 0,C 180,E1 -22740.37,E2 -22740.37} C_VEL
LIN {X 0,Y 189.296,Z 355.861,A -85,B 0,C 180,E1 -22742.349,E2 -22742.349} C_VEL
LIN {X 0,Y 186.67,Z 362.072,A -85,B 0,C 180,E1 -22744.344,E2 -22744.344} C_VEL
LIN {X 0,Y 184.431,Z 367.186,A -85,B 0,C 180,E1 -22746.362,E2 -22746.362} C_VEL
LIN {X 0,Y 182.544,Z 371.688,A -85,B 0,C 180,E1 -22748.546,E2 -22748.546} C_VEL
LIN {X 0,Y 180.03,Z 376.926,A -85,B 0,C 180,E1 -22751.802,E2 -22751.802} C_VEL
LIN {X 0,Y 178.102,Z 380.84,A -85,B 0,C 180,E1 -22755.138,E2 -22755.138} C_VEL
LIN {X 0,Y 176.952,Z 383.536,A -85,B 0,C 180,E1 -22758.546,E2 -22758.546} C_VEL
LIN {X 0,Y 176.482,Z 384.631,A -85,B 0,C 180,E1 -22760.835,E2 -22760.835} C_VEL
LIN {X 0,Y 176.247,Z 385.246,A -85,B 0,C 180,E1 -22763.13,E2 -22763.13} C_VEL
LIN {X 0,Y 176.23,Z 385.395,A -85,B 0,C 180,E1 -22765.557,E2 -22765.557} C_VEL
LIN {X 0,Y 176.443,Z 385.112,A -85,B 0,C 180,E1 -22767.718,E2 -22767.718} C_VEL
LIN {X 0,Y 176.571,Z 384.256,A -85,B 0,C 180,E1 -22770,E2 -22770} C_VEL
LIN {X 0,Y 176.604,Z 382.741,A -85,B 0,C 180,E1 -22772.351,E2 -22772.351} C_VEL
LIN {X 0,Y 175.941,Z 381.689,A -85,B 0,C 180,E1 -22773.595,E2 -22773.595} C_VEL
LIN {X 0,Y 173.296,Z 379.565,A -85,B 0,C 180,E1 -22775.555,E2 -22775.555} C_VEL
LIN {X 0,Y 170.699,Z 378.232,A -85,B 0,C 180,E1 -22777.583,E2 -22777.583} C_VEL
LIN {X 0,Y 170.103,Z 378.489,A -85,B 0,C 180,E1 -22778.892,E2 -22778.892} C_VEL
LIN {X 0,Y 170.486,Z 380.234,A -85,B 0,C 180,E1 -22781.895,E2 -22781.895} C_VEL
LIN {X 0,Y 172.162,Z 381.974,A -85,B 0,C 180,E1 -22786.604,E2 -22786.604} C_VEL
LIN {X 0,Y 175.401,Z 382.595,A -85,B 0,C 180,E1 -22791.138,E2 -22791.138} C_VEL
LIN {X 0,Y 179.89,Z 382.082,A -85,B 0,C 180,E1 -22795.452,E2 -22795.452} C_VEL
LIN {X 0,Y 185.577,Z 380.459,A -85,B 0,C 180,E1 -22799.494,E2 -22799.494} C_VEL
LIN {X 0,Y 192.577,Z 377.738,A -85,B 0,C 180,E1 -22803.191,E2 -22803.191} C_VEL
LIN {X 0,Y 200.76,Z 373.872,A -85,B 0,C 180,E1 -22806.522,E2 -22806.522} C_VEL
LIN {X 0,Y 209.635,Z 368.856,A -85,B 0,C 180,E1 -22809.567,E2 -22809.567} C_VEL
LIN {X 0,Y 214.196,Z 365.251,A -85,B 0,C 180,E1 -22812.271,E2 -22812.271} C_VEL
LIN {X 0,Y 215.516,Z 364.1,A -85,B 0,C 180,E1 -22813.222,E2 -22813.222} C_VEL
LIN {X 0,Y 216.739,Z 362.928,A -85,B 0,C 180,E1 -22814.49,E2 -22814.49} C_VEL
LIN {X 0,Y 217.69,Z 361.545,A -85,B 0,C 180,E1 -22817.315,E2 -22817.315} C_VEL
LIN {X 0,Y 217.695,Z 361.166,A -85,B 0,C 180,E1 -22819.784,E2 -22819.784} C_VEL
LIN {X 0,Y 217.158,Z 361.446,A -85,B 0,C 180,E1 -22822.055,E2 -22822.055} C_VEL
LIN {X 0,Y 213.596,Z 363.324,A -85,B 0,C 180,E1 -22823.683,E2 -22823.683} C_VEL
LIN {X 0,Y 204.602,Z 367.322,A -85,B 0,C 180,E1 -22826.661,E2 -22826.661} C_VEL
LIN {X 0,Y 196.422,Z 370.045,A -85,B 0,C 180,E1 -22829.939,E2 -22829.939} C_VEL
LIN {X 0,Y 189.217,Z 371.514,A -85,B 0,C 180,E1 -22833.531,E2 -22833.531} C_VEL
LIN {X 0,Y 182.974,Z 371.793,A -85,B 0,C 180,E1 -22837.412,E2 -22837.412} C_VEL
LIN {X 0,Y 177.923,Z 370.847,A -85,B 0,C 180,E1 -22841.579,E2 -22841.579} C_VEL
LIN {X 0,Y 175.74,Z 369.916,A -85,B 0,C 180,E1 -22843.744,E2 -22843.744} C_VEL
LIN {X 0,Y 172.788,Z 367.134,A -85,B 0,C 180,E1 -22848.266,E2 -22848.266} C_VEL
LIN {X 0,Y 170.904,Z 363.039,A -85,B 0,C 180,E1 -22852.914,E2 -22852.914} C_VEL
LIN {X 0,Y 169.733,Z 357.442,A -85,B 0,C 180,E1 -22857.627,E2 -22857.627} C_VEL
LIN {X 0,Y 169.589,Z 352.182,A -85,B 0,C 180,E1 -22861.188,E2 -22861.188} C_VEL
LIN {X 0,Y 169.735,Z 344.713,A -85,B 0,C 180,E1 -22865.286,E2 -22865.286} C_VEL
LIN {X 0,Y 170.205,Z 336.602,A -85,B 0,C 180,E1 -22868.908,E2 -22868.908} C_VEL
LIN {X 0,Y 170.92,Z 326.821,A -85,B 0,C 180,E1 -22872.467,E2 -22872.467} C_VEL
LIN {X 0,Y 172.116,Z 316.053,A -85,B 0,C 180,E1 -22875.695,E2 -22875.695} C_VEL
LIN {X 0,Y 173.386,Z 303.961,A -85,B 0,C 180,E1 -22878.615,E2 -22878.615} C_VEL
LIN {X 0,Y 174.418,Z 293.758,A -85,B 0,C 180,E1 -22880.645,E2 -22880.645} C_VEL
LIN {X 0,Y 172.286,Z 281.469,A -85,B 0,C 180,E1 -22882.642,E2 -22882.642} C_VEL
LIN {X 0,Y 170.13,Z 267.294,A -85,B 0,C 180,E1 -22884.48,E2 -22884.48} C_VEL
LIN {X 0,Y 170.593,Z 267.234,A -85,B 0,C 180,E1 -22890.099,E2 -22890.099} C_VEL
LIN {X 0,Y 171.054,Z 267.173,A -85,B 0,C 180,E1 -22895.115,E2 -22895.115} C_VEL
LIN {X 0,Y 171.286,Z 267.15,A -85,B 0,C 180,E1 -22898.776,E2 -22898.776} C_VEL
LIN {X 0,Y 171.334,Z 267.141,A -85,B 0,C 180,E1 -22902.408,E2 -22902.408} C_VEL
LIN {X 0,Y 171.335,Z 267.14,A -85,B 0,C 180,E1 -22907.591,E2 -22907.591} C_VEL
LIN {X 0,Y 171.362,Z 267.14,A -85,B 0,C 180,E1 -22912.034,E2 -22912.034} C_VEL
LIN {X 0,Y 171.4,Z 267.137,A -85,B 0,C 180,E1 -22915.093,E2 -22915.093} C_VEL
LIN {X 0,Y 171.412,Z 267.134,A -85,B 0,C 180,E1 -22920.527,E2 -22920.527} C_VEL
LIN {X 0,Y 171.445,Z 267.129,A -85,B 0,C 180,E1 -22925.799,E2 -22925.799} C_VEL
LIN {X 0,Y 171.582,Z 267.108,A -85,B 0,C 180,E1 -22930.871,E2 -22930.871} C_VEL
LIN {X 0,Y 171.58,Z 267.113,A -85,B 0,C 180,E1 -22935.773,E2 -22935.773} C_VEL
LIN {X 0,Y 171.846,Z 267.082,A -85,B 0,C 180,E1 -22940.584,E2 -22940.584} C_VEL
LIN {X 0,Y 171.803,Z 267.099,A -85,B 0,C 180,E1 -22945.601,E2 -22945.601} C_VEL
LIN {X 0,Y 172.858,Z 270.664,A -85,B 0,C 180,E1 -22948.835,E2 -22948.835} C_VEL
LIN {X 0,Y 173.184,Z 273.461,A -85,B 0,C 180,E1 -22951.162,E2 -22951.162} C_VEL
LIN {X 0,Y 172.937,Z 277.827,A -85,B 0,C 180,E1 -22954.662,E2 -22954.662} C_VEL
LIN {X 0,Y 172.201,Z 284.39,A -85,B 0,C 180,E1 -22959.757,E2 -22959.757} C_VEL
LIN {X 0,Y 174.353,Z 295.437,A -85,B 0,C 180,E1 -22960.992,E2 -22960.992} C_VEL
LIN {X 0,Y 175.705,Z 304.458,A -85,B 0,C 180,E1 -22962.257,E2 -22962.257} C_VEL
LIN {X 0,Y 176.899,Z 315.017,A -85,B 0,C 180,E1 -22964.083,E2 -22964.083} C_VEL
LIN {X 0,Y 177.057,Z 319.201,A -85,B 0,C 180,E1 -22964.952,E2 -22964.952} C_VEL
LIN {X 0,Y 175.616,Z 327.964,A -85,B 0,C 180,E1 -22966.864,E2 -22966.864} C_VEL
LIN {X 0,Y 173.907,Z 337.339,A -85,B 0,C 180,E1 -22969.475,E2 -22969.475} C_VEL
LIN {X 0,Y 172.48,Z 344.716,A -85,B 0,C 180,E1 -22972.142,E2 -22972.142} C_VEL
LIN {X 0,Y 171.353,Z 350.571,A -85,B 0,C 180,E1 -22974.766,E2 -22974.766} C_VEL
LIN {X 0,Y 170.397,Z 355.666,A -85,B 0,C 180,E1 -22977.613,E2 -22977.613} C_VEL
LIN {X 0,Y 169.46,Z 360.663,A -85,B 0,C 180,E1 -22981.226,E2 -22981.226} C_VEL
LIN {X 0,Y 169.071,Z 363.214,A -85,B 0,C 180,E1 -22983.76,E2 -22983.76} C_VEL
LIN {X 0,Y 169.027,Z 365.999,A -85,B 0,C 180,E1 -22987.814,E2 -22987.814} C_VEL
LIN {X 0,Y 169.521,Z 367.272,A -85,B 0,C 180,E1 -22991.733,E2 -22991.733} C_VEL
LIN {X 0,Y 170.617,Z 367.283,A -85,B 0,C 180,E1 -22995.552,E2 -22995.552} C_VEL
LIN {X 0,Y 172.259,Z 366.03,A -85,B 0,C 180,E1 -22999.247,E2 -22999.247} C_VEL
LIN {X 0,Y 174.922,Z 362.829,A -85,B 0,C 180,E1 -23003.471,E2 -23003.471} C_VEL
LIN {X 0,Y 177.237,Z 359.477,A -85,B 0,C 180,E1 -23006.379,E2 -23006.379} C_VEL
LIN {X 0,Y 180.307,Z 354.473,A -85,B 0,C 180,E1 -23009.554,E2 -23009.554} C_VEL
LIN {X 0,Y 183.853,Z 347.92,A -85,B 0,C 180,E1 -23012.534,E2 -23012.534} C_VEL
LIN {X 0,Y 186.703,Z 342.064,A -85,B 0,C 180,E1 -23014.612,E2 -23014.612} C_VEL
LIN {X 0,Y 189.412,Z 335.587,A -85,B 0,C 180,E1 -23016.493,E2 -23016.493} C_VEL
LIN {X 0,Y 190.043,Z 330.923,A -85,B 0,C 180,E1 -23017.969,E2 -23017.969} C_VEL
LIN {X 0,Y 190.152,Z 324.167,A -85,B 0,C 180,E1 -23020.008,E2 -23020.008} C_VEL
LIN {X 0,Y 189.547,Z 316.663,A -85,B 0,C 180,E1 -23022.188,E2 -23022.188} C_VEL
LIN {X 0,Y 188.24,Z 309.285,A -85,B 0,C 180,E1 -23024.295,E2 -23024.295} C_VEL
LIN {X 0,Y 186.731,Z 304.587,A -85,B 0,C 180,E1 -23025.77,E2 -23025.77} C_VEL
LIN {X 0,Y 184.138,Z 299.147,A -85,B 0,C 180,E1 -23027.744,E2 -23027.744} C_VEL
LIN {X 0,Y 182.523,Z 296.312,A -85,B 0,C 180,E1 -23028.9,E2 -23028.9} C_VEL
LIN {X 0,Y 180.119,Z 292.134,A -85,B 0,C 180,E1 -23030.596,E2 -23030.596} C_VEL
LIN {X 0,Y 177.59,Z 288.137,A -85,B 0,C 180,E1 -23032.396,E2 -23032.396} C_VEL
LIN {X 0,Y 177.363,Z 287.59,A -85,B 0,C 180,E1 -23032.601,E2 -23032.601} C_VEL
LIN {X 0,Y 177.047,Z 284.146,A -85,B 0,C 180,E1 -23037.725,E2 -23037.725} C_VEL
LIN {X 0,Y 176.963,Z 282.757,A -85,B 0,C 180,E1 -23040,E2 -23040} C_VEL
LIN {X 0,Y 176.747,Z 281.622,A -85,B 0,C 180,E1 -23042.279,E2 -23042.279} C_VEL
LIN {X 0,Y 176.035,Z 279.907,A -85,B 0,C 180,E1 -23046.879,E2 -23046.879} C_VEL
LIN {X 0,Y 175.666,Z 278.657,A -85,B 0,C 180,E1 -23051.539,E2 -23051.539} C_VEL
LIN {X 0,Y 175.375,Z 278.132,A -85,B 0,C 180,E1 -23056.291,E2 -23056.291} C_VEL
LIN {X 0,Y 175.471,Z 278.297,A -85,B 0,C 180,E1 -23061.129,E2 -23061.129} C_VEL
LIN {X 0,Y 175.915,Z 279.264,A -85,B 0,C 180,E1 -23066.069,E2 -23066.069} C_VEL
LIN {X 0,Y 176.678,Z 281.246,A -85,B 0,C 180,E1 -23071.139,E2 -23071.139} C_VEL
LIN {X 0,Y 177.954,Z 284.405,A -85,B 0,C 180,E1 -23076.327,E2 -23076.327} C_VEL
LIN {X 0,Y 179.234,Z 287.703,A -85,B 0,C 180,E1 -23080.315,E2 -23080.315} C_VEL
LIN {X 0,Y 180.253,Z 290.421,A -85,B 0,C 180,E1 -23083.024,E2 -23083.024} C_VEL
LIN {X 0,Y 181.148,Z 294.752,A -85,B 0,C 180,E1 -23086.278,E2 -23086.278} C_VEL
LIN {X 0,Y 184.002,Z 299.944,A -85,B 0,C 180,E1 -23088.056,E2 -23088.056} C_VEL
LIN {X 0,Y 186.079,Z 305.708,A -85,B 0,C 180,E1 -23089.504,E2 -23089.504} C_VEL
LIN {X 0,Y 188.223,Z 315.236,A -85,B 0,C 180,E1 -23091.639,E2 -23091.639} C_VEL
LIN {X 0,Y 189.463,Z 325.682,A -85,B 0,C 180,E1 -23093.961,E2 -23093.961} C_VEL
LIN {X 0,Y 189.596,Z 331.912,A -85,B 0,C 180,E1 -23095.33,E2 -23095.33} C_VEL
LIN {X 0,Y 187.523,Z 341.948,A -85,B 0,C 180,E1 -23097.402,E2 -23097.402} C_VEL
LIN {X 0,Y 185.818,Z 349.365,A -85,B 0,C 180,E1 -23099.297,E2 -23099.297} C_VEL
LIN {X 0,Y 183.074,Z 356.583,A -85,B 0,C 180,E1 -23101.324,E2 -23101.324} C_VEL
LIN {X 0,Y 180.316,Z 362.614,A -85,B 0,C 180,E1 -23103.37,E2 -23103.37} C_VEL
LIN {X 0,Y 177.803,Z 367.898,A -85,B 0,C 180,E1 -23105.605,E2 -23105.605} C_VEL
LIN {X 0,Y 174.988,Z 373.812,A -85,B 0,C 180,E1 -23108.81,E2 -23108.81} C_VEL
LIN {X 0,Y 172.521,Z 378.439,A -85,B 0,C 180,E1 -23112.21,E2 -23112.21} C_VEL
LIN {X 0,Y 170.715,Z 381.713,A -85,B 0,C 180,E1 -23115.7,E2 -23115.7} C_VEL
LIN {X 0,Y 169.974,Z 383.32,A -85,B 0,C 180,E1 -23118.069,E2 -23118.069} C_VEL
LIN {X 0,Y 169.454,Z 384.385,A -85,B 0,C 180,E1 -23120.451,E2 -23120.451} C_VEL
LIN {X 0,Y 169.168,Z 384.902,A -85,B 0,C 180,E1 -23122.841,E2 -23122.841} C_VEL
LIN {X 0,Y 169.169,Z 384.94,A -85,B 0,C 180,E1 -23125.608,E2 -23125.608} C_VEL
LIN {X 0,Y 169.368,Z 384.587,A -85,B 0,C 180,E1 -23127.622,E2 -23127.622} C_VEL
LIN {X 0,Y 169.503,Z 383.695,A -85,B 0,C 180,E1 -23130,E2 -23130} C_VEL
LIN {X 0,Y 169.54,Z 381.19,A -85,B 0,C 180,E1 -23133.565,E2 -23133.565} C_VEL
LIN {X 0,Y 169.731,Z 379.313,A -85,B 0,C 180,E1 -23135.553,E2 -23135.553} C_VEL
LIN {X 0,Y 170.13,Z 377.369,A -85,B 0,C 180,E1 -23137.248,E2 -23137.248} C_VEL
LIN {X 0,Y 170.103,Z 378.489,A -85,B 0,C 180,E1 -23138.892,E2 -23138.892} C_VEL
LIN {X 0,Y 169.629,Z 379.558,A -85,B 0,C 180,E1 -23140.843,E2 -23140.843} C_VEL
LIN {X 0,Y 167.593,Z 380.522,A -85,B 0,C 180,E1 -23144.124,E2 -23144.124} C_VEL
LIN {X 0,Y 166.318,Z 380.977,A -85,B 0,C 180,E1 -23146.812,E2 -23146.812} C_VEL
LIN {X 0,Y 166.426,Z 381.336,A -85,B 0,C 180,E1 -23148.843,E2 -23148.843} C_VEL
LIN {X 0,Y 166.776,Z 381.478,A -85,B 0,C 180,E1 -23149.508,E2 -23149.508} C_VEL
LIN {X 0,Y 170.963,Z 381.928,A -85,B 0,C 180,E1 -23154.274,E2 -23154.274} C_VEL
LIN {X 0,Y 176.278,Z 381.234,A -85,B 0,C 180,E1 -23158.583,E2 -23158.583} C_VEL
LIN {X 0,Y 182.845,Z 379.475,A -85,B 0,C 180,E1 -23162.556,E2 -23162.556} C_VEL
LIN {X 0,Y 190.823,Z 376.625,A -85,B 0,C 180,E1 -23166.107,E2 -23166.107} C_VEL
LIN {X 0,Y 199.717,Z 372.643,A -85,B 0,C 180,E1 -23169.303,E2 -23169.303} C_VEL
LIN {X 0,Y 204.268,Z 370.281,A -85,B 0,C 180,E1 -23170.823,E2 -23170.823} C_VEL
LIN {X 0,Y 207.489,Z 368.12,A -85,B 0,C 180,E1 -23172.644,E2 -23172.644} C_VEL
LIN {X 0,Y 208.947,Z 367.064,A -85,B 0,C 180,E1 -23173.593,E2 -23173.593} C_VEL
LIN {X 0,Y 210.139,Z 366.113,A -85,B 0,C 180,E1 -23174.615,E2 -23174.615} C_VEL
LIN {X 0,Y 210.751,Z 365.512,A -85,B 0,C 180,E1 -23175.549,E2 -23175.549} C_VEL
LIN {X 0,Y 211.225,Z 364.864,A -85,B 0,C 180,E1 -23177.055,E2 -23177.055} C_VEL
LIN {X 0,Y 211.381,Z 364.52,A -85,B 0,C 180,E1 -23178.321,E2 -23178.321} C_VEL
LIN {X 0,Y 211.166,Z 364.356,A -85,B 0,C 180,E1 -23180.776,E2 -23180.776} C_VEL
LIN {X 0,Y 208.133,Z 365.666,A -85,B 0,C 180,E1 -23182.569,E2 -23182.569} C_VEL
LIN {X 0,Y 198.861,Z 369.126,A -85,B 0,C 180,E1 -23185.566,E2 -23185.566} C_VEL
LIN {X 0,Y 190.404,Z 371.375,A -85,B 0,C 180,E1 -23188.885,E2 -23188.885} C_VEL
LIN {X 0,Y 182.937,Z 372.427,A -85,B 0,C 180,E1 -23192.548,E2 -23192.548} C_VEL
LIN {X 0,Y 176.456,Z 372.28,A -85,B 0,C 180,E1 -23196.529,E2 -23196.529} C_VEL
LIN {X 0,Y 171.228,Z 370.92,A -85,B 0,C 180,E1 -23200.831,E2 -23200.831} C_VEL
LIN {X 0,Y 168.738,Z 369.64,A -85,B 0,C 180,E1 -23203.33,E2 -23203.33} C_VEL
LIN {X 0,Y 165.293,Z 365.66,A -85,B 0,C 180,E1 -23208.97,E2 -23208.97} C_VEL
LIN {X 0,Y 163.498,Z 360.832,A -85,B 0,C 180,E1 -23213.831,E2 -23213.831} C_VEL
LIN {X 0,Y 162.652,Z 354.496,A -85,B 0,C 180,E1 -23218.762,E2 -23218.762} C_VEL
LIN {X 0,Y 162.621,Z 347.451,A -85,B 0,C 180,E1 -23223.097,E2 -23223.097} C_VEL
LIN {X 0,Y 162.952,Z 339.66,A -85,B 0,C 180,E1 -23226.98,E2 -23226.98} C_VEL
LIN {X 0,Y 163.551,Z 331.044,A -85,B 0,C 180,E1 -23230.523,E2 -23230.523} C_VEL
LIN {X 0,Y 164.316,Z 322.059,A -85,B 0,C 180,E1 -23233.606,E2 -23233.606} C_VEL
LIN {X 0,Y 165.477,Z 311.377,A -85,B 0,C 180,E1 -23236.66,E2 -23236.66} C_VEL
LIN {X 0,Y 166.896,Z 298.237,A -85,B 0,C 180,E1 -23239.687,E2 -23239.687} C_VEL
LIN {X 0,Y 167.31,Z 294.042,A -85,B 0,C 180,E1 -23240.507,E2 -23240.507} C_VEL
LIN {X 0,Y 165.022,Z 280.944,A -85,B 0,C 180,E1 -23242.703,E2 -23242.703} C_VEL
LIN {X 0,Y 163.086,Z 268.172,A -85,B 0,C 180,E1 -23244.457,E2 -23244.457} C_VEL
LIN {X 0,Y 163.623,Z 268.103,A -85,B 0,C 180,E1 -23251.027,E2 -23251.027} C_VEL
LIN {X 0,Y 164.013,Z 268.051,A -85,B 0,C 180,E1 -23255.495,E2 -23255.495} C_VEL
LIN {X 0,Y 164.228,Z 268.025,A -85,B 0,C 180,E1 -23259.935,E2 -23259.935} C_VEL
LIN {X 0,Y 164.282,Z 268.024,A -85,B 0,C 180,E1 -23263.342,E2 -23263.342} C_VEL
LIN {X 0,Y 164.264,Z 268.022,A -85,B 0,C 180,E1 -23266.798,E2 -23266.798} C_VEL
LIN {X 0,Y 164.292,Z 268.022,A -85,B 0,C 180,E1 -23270.354,E2 -23270.354} C_VEL
LIN {X 0,Y 164.328,Z 268.014,A -85,B 0,C 180,E1 -23274.351,E2 -23274.351} C_VEL
LIN {X 0,Y 164.369,Z 268.009,A -85,B 0,C 180,E1 -23279.13,E2 -23279.13} C_VEL
LIN {X 0,Y 164.398,Z 268.008,A -85,B 0,C 180,E1 -23284.69,E2 -23284.69} C_VEL
LIN {X 0,Y 164.487,Z 267.996,A -85,B 0,C 180,E1 -23290.051,E2 -23290.051} C_VEL
LIN {X 0,Y 164.527,Z 267.991,A -85,B 0,C 180,E1 -23295.149,E2 -23295.149} C_VEL
LIN {X 0,Y 164.768,Z 267.963,A -85,B 0,C 180,E1 -23300.176,E2 -23300.176} C_VEL
LIN {X 0,Y 164.751,Z 267.964,A -85,B 0,C 180,E1 -23304.722,E2 -23304.722} C_VEL
LIN {X 0,Y 165.963,Z 272.328,A -85,B 0,C 180,E1 -23308.786,E2 -23308.786} C_VEL
LIN {X 0,Y 166.253,Z 275.112,A -85,B 0,C 180,E1 -23311.211,E2 -23311.211} C_VEL
LIN {X 0,Y 165.92,Z 279.584,A -85,B 0,C 180,E1 -23314.859,E2 -23314.859} C_VEL
LIN {X 0,Y 165.322,Z 284.663,A -85,B 0,C 180,E1 -23318.941,E2 -23318.941} C_VEL
LIN {X 0,Y 167.6,Z 296.482,A -85,B 0,C 180,E1 -23320.342,E2 -23320.342} C_VEL
LIN {X 0,Y 168.911,Z 305.705,A -85,B 0,C 180,E1 -23321.703,E2 -23321.703} C_VEL
LIN {X 0,Y 170.064,Z 316.727,A -85,B 0,C 180,E1 -23323.746,E2 -23323.746} C_VEL
LIN {X 0,Y 170.002,Z 320.986,A -85,B 0,C 180,E1 -23324.667,E2 -23324.667} C_VEL
LIN {X 0,Y 168.226,Z 330.85,A -85,B 0,C 180,E1 -23327.004,E2 -23327.004} C_VEL
LIN {X 0,Y 166.946,Z 337.611,A -85,B 0,C 180,E1 -23329.041,E2 -23329.041} C_VEL
LIN {X 0,Y 165.506,Z 344.823,A -85,B 0,C 180,E1 -23331.741,E2 -23331.741} C_VEL
LIN {X 0,Y 164.522,Z 349.7,A -85,B 0,C 180,E1 -23333.942,E2 -23333.942} C_VEL
LIN {X 0,Y 163.466,Z 355.027,A -85,B 0,C 180,E1 -23336.913,E2 -23336.913} C_VEL
LIN {X 0,Y 162.565,Z 359.587,A -85,B 0,C 180,E1 -23340.157,E2 -23340.157} C_VEL
LIN {X 0,Y 162.095,Z 362.486,A -85,B 0,C 180,E1 -23342.817,E2 -23342.817} C_VEL
LIN {X 0,Y 161.88,Z 364.991,A -85,B 0,C 180,E1 -23345.879,E2 -23345.879} C_VEL
LIN {X 0,Y 161.983,Z 366.567,A -85,B 0,C 180,E1 -23348.65,E2 -23348.65} C_VEL
LIN {X 0,Y 162.207,Z 367.34,A -85,B 0,C 180,E1 -23350.535,E2 -23350.535} C_VEL
LIN {X 0,Y 162.876,Z 367.884,A -85,B 0,C 180,E1 -23353.661,E2 -23353.661} C_VEL
LIN {X 0,Y 163.966,Z 367.634,A -85,B 0,C 180,E1 -23356.774,E2 -23356.774} C_VEL
LIN {X 0,Y 165.752,Z 366.223,A -85,B 0,C 180,E1 -23360.504,E2 -23360.504} C_VEL
LIN {X 0,Y 167.304,Z 364.66,A -85,B 0,C 180,E1 -23362.953,E2 -23362.953} C_VEL
LIN {X 0,Y 170.361,Z 360.751,A -85,B 0,C 180,E1 -23366.841,E2 -23366.841} C_VEL
LIN {X 0,Y 173.422,Z 356.16,A -85,B 0,C 180,E1 -23370.048,E2 -23370.048} C_VEL
LIN {X 0,Y 177.169,Z 350.005,A -85,B 0,C 180,E1 -23373.194,E2 -23373.194} C_VEL
LIN {X 0,Y 180.936,Z 342.757,A -85,B 0,C 180,E1 -23375.895,E2 -23375.895} C_VEL
LIN {X 0,Y 183.702,Z 336.427,A -85,B 0,C 180,E1 -23377.803,E2 -23377.803} C_VEL
LIN {X 0,Y 184.323,Z 330.172,A -85,B 0,C 180,E1 -23379.93,E2 -23379.93} C_VEL
LIN {X 0,Y 184.316,Z 322.362,A -85,B 0,C 180,E1 -23382.412,E2 -23382.412} C_VEL
LIN {X 0,Y 183.386,Z 314.088,A -85,B 0,C 180,E1 -23384.983,E2 -23384.983} C_VEL
LIN {X 0,Y 182.17,Z 309.273,A -85,B 0,C 180,E1 -23386.616,E2 -23386.616} C_VEL
LIN {X 0,Y 178.849,Z 301.934,A -85,B 0,C 180,E1 -23389.612,E2 -23389.612} C_VEL
LIN {X 0,Y 176.743,Z 297.919,A -85,B 0,C 180,E1 -23391.388,E2 -23391.388} C_VEL
LIN {X 0,Y 174.053,Z 293.308,A -85,B 0,C 180,E1 -23393.624,E2 -23393.624} C_VEL
LIN {X 0,Y 171.564,Z 289.939,A -85,B 0,C 180,E1 -23395.668,E2 -23395.668} C_VEL
LIN {X 0,Y 170.749,Z 288.142,A -85,B 0,C 180,E1 -23396.608,E2 -23396.608} C_VEL
LIN {X 0,Y 170.706,Z 286.154,A -85,B 0,C 180,E1 -23400,E2 -23400} C_VEL
LIN {X 0,Y 170.526,Z 285.038,A -85,B 0,C 180,E1 -23402.362,E2 -23402.362} C_VEL
LIN {X 0,Y 169.894,Z 283.41,A -85,B 0,C 180,E1 -23407.129,E2 -23407.129} C_VEL
LIN {X 0,Y 169.586,Z 282.315,A -85,B 0,C 180,E1 -23411.959,E2 -23411.959} C_VEL
LIN {X 0,Y 169.375,Z 281.982,A -85,B 0,C 180,E1 -23416.885,E2 -23416.885} C_VEL
LIN {X 0,Y 169.591,Z 282.338,A -85,B 0,C 180,E1 -23421.899,E2 -23421.899} C_VEL
LIN {X 0,Y 170.14,Z 283.568,A -85,B 0,C 180,E1 -23427.025,E2 -23427.025} C_VEL
LIN {X 0,Y 171.076,Z 285.906,A -85,B 0,C 180,E1 -23432.28,E2 -23432.28} C_VEL
LIN {X 0,Y 172.502,Z 289.506,A -85,B 0,C 180,E1 -23437.671,E2 -23437.671} C_VEL
LIN {X 0,Y 174.228,Z 294.007,A -85,B 0,C 180,E1 -23442.628,E2 -23442.628} C_VEL
LIN {X 0,Y 178.16,Z 301.112,A -85,B 0,C 180,E1 -23445.568,E2 -23445.568} C_VEL
LIN {X 0,Y 180.672,Z 306.168,A -85,B 0,C 180,E1 -23447.349,E2 -23447.349} C_VEL
LIN {X 0,Y 182.016,Z 311.432,A -85,B 0,C 180,E1 -23448.757,E2 -23448.757} C_VEL
LIN {X 0,Y 183.735,Z 322.609,A -85,B 0,C 180,E1 -23451.435,E2 -23451.435} C_VEL
LIN {X 0,Y 184.004,Z 332.06,A -85,B 0,C 180,E1 -23453.709,E2 -23453.709} C_VEL
LIN {X 0,Y 183.578,Z 335.281,A -85,B 0,C 180,E1 -23454.44,E2 -23454.44} C_VEL
LIN {X 0,Y 181.679,Z 343.269,A -85,B 0,C 180,E1 -23456.215,E2 -23456.215} C_VEL
LIN {X 0,Y 179.173,Z 352.317,A -85,B 0,C 180,E1 -23458.686,E2 -23458.686} C_VEL
LIN {X 0,Y 175.456,Z 360.399,A -85,B 0,C 180,E1 -23461.271,E2 -23461.271} C_VEL
LIN {X 0,Y 171.992,Z 367.036,A -85,B 0,C 180,E1 -23464.023,E2 -23464.023} C_VEL
LIN {X 0,Y 169.362,Z 372.152,A -85,B 0,C 180,E1 -23466.783,E2 -23466.783} C_VEL
LIN {X 0,Y 167.47,Z 375.586,A -85,B 0,C 180,E1 -23469.102,E2 -23469.102} C_VEL
LIN {X 0,Y 164.995,Z 379.605,A -85,B 0,C 180,E1 -23472.653,E2 -23472.653} C_VEL
LIN {X 0,Y 163.798,Z 381.579,A -85,B 0,C 180,E1 -23475.082,E2 -23475.082} C_VEL
LIN {X 0,Y 162.981,Z 383.076,A -85,B 0,C 180,E1 -23477.549,E2 -23477.549} C_VEL
LIN {X 0,Y 162.422,Z 384.105,A -85,B 0,C 180,E1 -23480.033,E2 -23480.033} C_VEL
LIN {X 0,Y 162.117,Z 384.562,A -85,B 0,C 180,E1 -23482.528,E2 -23482.528} C_VEL
LIN {X 0,Y 162.108,Z 384.483,A -85,B 0,C 180,E1 -23485.663,E2 -23485.663} C_VEL
LIN {X 0,Y 162.294,Z 384.049,A -85,B 0,C 180,E1 -23487.518,E2 -23487.518} C_VEL
LIN {X 0,Y 162.436,Z 383.076,A -85,B 0,C 180,E1 -23490,E2 -23490} C_VEL
LIN {X 0,Y 162.484,Z 381.537,A -85,B 0,C 180,E1 -23492.479,E2 -23492.479} C_VEL
LIN {X 0,Y 162.792,Z 378.051,A -85,B 0,C 180,E1 -23496.196,E2 -23496.196} C_VEL
LIN {X 0,Y 163.225,Z 376.042,A -85,B 0,C 180,E1 -23497.982,E2 -23497.982} C_VEL
LIN {X 0,Y 163.651,Z 378.863,A -85,B 0,C 180,E1 -23502.4,E2 -23502.4} C_VEL
LIN {X 0,Y 165.425,Z 380.916,A -85,B 0,C 180,E1 -23507.301,E2 -23507.301} C_VEL
LIN {X 0,Y 166.776,Z 381.478,A -85,B 0,C 180,E1 -23509.508,E2 -23509.508} C_VEL
LIN {X 0,Y 167.601,Z 381.813,A -85,B 0,C 180,E1 -23511.511,E2 -23511.511} C_VEL
LIN {X 0,Y 167.832,Z 381.76,A -85,B 0,C 180,E1 -23514.898,E2 -23514.898} C_VEL
LIN {X 0,Y 168.42,Z 381.355,A -85,B 0,C 180,E1 -23517.591,E2 -23517.591} C_VEL
LIN {X 0,Y 169.898,Z 380.949,A -85,B 0,C 180,E1 -23519.521,E2 -23519.521} C_VEL
LIN {X 0,Y 170.684,Z 380.806,A -85,B 0,C 180,E1 -23520.126,E2 -23520.126} C_VEL
LIN {X 0,Y 176.918,Z 379.546,A -85,B 0,C 180,E1 -23523.79,E2 -23523.79} C_VEL
LIN {X 0,Y 185.159,Z 377.139,A -85,B 0,C 180,E1 -23527.396,E2 -23527.396} C_VEL
LIN {X 0,Y 195.859,Z 372.982,A -85,B 0,C 180,E1 -23531.102,E2 -23531.102} C_VEL
LIN {X 0,Y 198.949,Z 371.56,A -85,B 0,C 180,E1 -23532.16,E2 -23532.16} C_VEL
LIN {X 0,Y 202.257,Z 369.655,A -85,B 0,C 180,E1 -23534.025,E2 -23534.025} C_VEL
LIN {X 0,Y 204.389,Z 368.079,A -85,B 0,C 180,E1 -23536.228,E2 -23536.228} C_VEL
LIN {X 0,Y 204.828,Z 367.254,A -85,B 0,C 180,E1 -23539.313,E2 -23539.313} C_VEL
LIN {X 0,Y 202.734,Z 367.858,A -85,B 0,C 180,E1 -23541.392,E2 -23541.392} C_VEL
LIN {X 0,Y 193.176,Z 370.795,A -85,B 0,C 180,E1 -23544.402,E2 -23544.402} C_VEL
LIN {X 0,Y 184.446,Z 372.562,A -85,B 0,C 180,E1 -23547.762,E2 -23547.762} C_VEL
LIN {X 0,Y 176.702,Z 373.164,A -85,B 0,C 180,E1 -23551.492,E2 -23551.492} C_VEL
LIN {X 0,Y 169.984,Z 372.607,A -85,B 0,C 180,E1 -23555.578,E2 -23555.578} C_VEL
LIN {X 0,Y 163.99,Z 370.579,A -85,B 0,C 180,E1 -23560.536,E2 -23560.536} C_VEL
LIN {X 0,Y 160.389,Z 367.92,A -85,B 0,C 180,E1 -23564.757,E2 -23564.757} C_VEL
LIN {X 0,Y 157.827,Z 363.759,A -85,B 0,C 180,E1 -23569.74,E2 -23569.74} C_VEL
LIN {X 0,Y 156.525,Z 359.76,A -85,B 0,C 180,E1 -23573.555,E2 -23573.555} C_VEL
LIN {X 0,Y 155.681,Z 352.998,A -85,B 0,C 180,E1 -23578.707,E2 -23578.707} C_VEL
LIN {X 0,Y 155.668,Z 345.584,A -85,B 0,C 180,E1 -23583.235,E2 -23583.235} C_VEL
LIN {X 0,Y 155.991,Z 338.119,A -85,B 0,C 180,E1 -23586.961,E2 -23586.961} C_VEL
LIN {X 0,Y 156.562,Z 330.049,A -85,B 0,C 180,E1 -23590.344,E2 -23590.344} C_VEL
LIN {X 0,Y 157.571,Z 318.807,A -85,B 0,C 180,E1 -23594.201,E2 -23594.201} C_VEL
LIN {X 0,Y 158.708,Z 307.433,A -85,B 0,C 180,E1 -23597.392,E2 -23597.392} C_VEL
LIN {X 0,Y 160.125,Z 294.833,A -85,B 0,C 180,E1 -23600.221,E2 -23600.221} C_VEL
LIN {X 0,Y 158.48,Z 284.475,A -85,B 0,C 180,E1 -23602.086,E2 -23602.086} C_VEL
LIN {X 0,Y 156.45,Z 271.748,A -85,B 0,C 180,E1 -23603.984,E2 -23603.984} C_VEL
LIN {X 0,Y 156.047,Z 269.049,A -85,B 0,C 180,E1 -23604.393,E2 -23604.393} C_VEL
LIN {X 0,Y 156.616,Z 268.977,A -85,B 0,C 180,E1 -23611.502,E2 -23611.502} C_VEL
LIN {X 0,Y 157.004,Z 268.926,A -85,B 0,C 180,E1 -23616.317,E2 -23616.317} C_VEL
LIN {X 0,Y 157.15,Z 268.907,A -85,B 0,C 180,E1 -23620.511,E2 -23620.511} C_VEL
LIN {X 0,Y 157.18,Z 268.906,A -85,B 0,C 180,E1 -23625.677,E2 -23625.677} C_VEL
LIN {X 0,Y 157.2,Z 268.905,A -85,B 0,C 180,E1 -23631.251,E2 -23631.251} C_VEL
LIN {X 0,Y 157.276,Z 268.893,A -85,B 0,C 180,E1 -23634.484,E2 -23634.484} C_VEL
LIN {X 0,Y 157.282,Z 268.892,A -85,B 0,C 180,E1 -23638.104,E2 -23638.104} C_VEL
LIN {X 0,Y 157.312,Z 268.889,A -85,B 0,C 180,E1 -23643.464,E2 -23643.464} C_VEL
LIN {X 0,Y 157.395,Z 268.879,A -85,B 0,C 180,E1 -23649.669,E2 -23649.669} C_VEL
LIN {X 0,Y 157.457,Z 268.869,A -85,B 0,C 180,E1 -23654.466,E2 -23654.466} C_VEL
LIN {X 0,Y 157.69,Z 268.846,A -85,B 0,C 180,E1 -23659.73,E2 -23659.73} C_VEL
LIN {X 0,Y 157.712,Z 268.904,A -85,B 0,C 180,E1 -23663.924,E2 -23663.924} C_VEL
LIN {X 0,Y 159.047,Z 273.958,A -85,B 0,C 180,E1 -23668.734,E2 -23668.734} C_VEL
LIN {X 0,Y 159.306,Z 276.815,A -85,B 0,C 180,E1 -23671.264,E2 -23671.264} C_VEL
LIN {X 0,Y 158.898,Z 281.342,A -85,B 0,C 180,E1 -23675.075,E2 -23675.075} C_VEL
LIN {X 0,Y 158.432,Z 285.195,A -85,B 0,C 180,E1 -23678.128,E2 -23678.128} C_VEL
LIN {X 0,Y 160.436,Z 295.562,A -85,B 0,C 180,E1 -23679.375,E2 -23679.375} C_VEL
LIN {X 0,Y 161.742,Z 303.977,A -85,B 0,C 180,E1 -23680.642,E2 -23680.642} C_VEL
LIN {X 0,Y 162.716,Z 312.335,A -85,B 0,C 180,E1 -23682.155,E2 -23682.155} C_VEL
LIN {X 0,Y 163.296,Z 319.534,A -85,B 0,C 180,E1 -23683.692,E2 -23683.692} C_VEL
LIN {X 0,Y 161.961,Z 327.608,A -85,B 0,C 180,E1 -23685.572,E2 -23685.572} C_VEL
LIN {X 0,Y 160.404,Z 335.571,A -85,B 0,C 180,E1 -23687.86,E2 -23687.86} C_VEL
LIN {X 0,Y 158.774,Z 343.571,A -85,B 0,C 180,E1 -23690.739,E2 -23690.739} C_VEL
LIN {X 0,Y 157.478,Z 349.939,A -85,B 0,C 180,E1 -23693.681,E2 -23693.681} C_VEL
LIN {X 0,Y 156.397,Z 355.174,A -85,B 0,C 180,E1 -23696.703,E2 -23696.703} C_VEL
LIN {X 0,Y 155.537,Z 359.444,A -85,B 0,C 180,E1 -23699.804,E2 -23699.804} C_VEL
LIN {X 0,Y 154.994,Z 362.814,A -85,B 0,C 180,E1 -23702.965,E2 -23702.965} C_VEL
LIN {X 0,Y 154.794,Z 365.345,A -85,B 0,C 180,E1 -23706.173,E2 -23706.173} C_VEL
LIN {X 0,Y 154.971,Z 367.136,A -85,B 0,C 180,E1 -23709.559,E2 -23709.559} C_VEL
LIN {X 0,Y 155.806,Z 368.21,A -85,B 0,C 180,E1 -23713.803,E2 -23713.803} C_VEL
LIN {X 0,Y 157.281,Z 367.982,A -85,B 0,C 180,E1 -23717.912,E2 -23717.912} C_VEL
LIN {X 0,Y 159.686,Z 366.116,A -85,B 0,C 180,E1 -23722.392,E2 -23722.392} C_VEL
LIN {X 0,Y 162.082,Z 363.658,A -85,B 0,C 180,E1 -23725.688,E2 -23725.688} C_VEL
LIN {X 0,Y 164.595,Z 360.502,A -85,B 0,C 180,E1 -23728.647,E2 -23728.647} C_VEL
LIN {X 0,Y 168.429,Z 355.19,A -85,B 0,C 180,E1 -23732.222,E2 -23732.222} C_VEL
LIN {X 0,Y 172.426,Z 348.685,A -85,B 0,C 180,E1 -23735.314,E2 -23735.314} C_VEL
LIN {X 0,Y 175.787,Z 342.519,A -85,B 0,C 180,E1 -23737.577,E2 -23737.577} C_VEL
LIN {X 0,Y 177.316,Z 339.462,A -85,B 0,C 180,E1 -23738.568,E2 -23738.568} C_VEL
LIN {X 0,Y 178.15,Z 335.853,A -85,B 0,C 180,E1 -23739.807,E2 -23739.807} C_VEL
LIN {X 0,Y 178.74,Z 329.352,A -85,B 0,C 180,E1 -23742.108,E2 -23742.108} C_VEL
LIN {X 0,Y 178.714,Z 322.453,A -85,B 0,C 180,E1 -23744.454,E2 -23744.454} C_VEL
LIN {X 0,Y 178.19,Z 316.995,A -85,B 0,C 180,E1 -23746.311,E2 -23746.311} C_VEL
LIN {X 0,Y 177.313,Z 313.308,A -85,B 0,C 180,E1 -23747.699,E2 -23747.699} C_VEL
LIN {X 0,Y 175.029,Z 307.657,A -85,B 0,C 180,E1 -23750.21,E2 -23750.21} C_VEL
